///////////////////////////////////////////////////////////////////////////////
// --- Finalizar
      JU    Final_EventoRecibido_DIDO;  // Finalizar



NETWORK
TITLE = ---- Accion del Evento --> Notificacion de Cambio de Estado de Trabajo del CBOX
///////////////////////////////////////////////////////////////////////////////
///////////////////////////////////////////////////////////////////////////////
// --- Tipo CBOX
DispositivoCBOX_EventoRecibido_DIDO:NOP   0;
      L     #AtributosDeDispositivos.Numero;  // Comprobacion del numero de CCPIF
      L     100;
      /I;
      L     "CTE_OffsetCCPIF";
      -I;
      L     1;
      <>I;  // Numero de CCPIF incorrecto
      JC    Final_EventoRecibido_DIDO;

      L     #AtributosDeDispositivos.Numero;  // Calculo del numero de CBOX
      L     100;
      MOD;  // Var verlo en la DB_Dispositivos
      T     #VarTempDispositivos.Numero;

      L     #VarTempDispositivos.Numero;  // Comprobacion del numero de CBOX
      L     1;  // Es menor de 1
      <I;  // No es correcto el numero de CBOX
      JC    Final_EventoRecibido_DIDO;
      L     #VarTempDispositivos.Numero;
      L     "CTE_MaxDispositivos";  // Si es mayor que el parametro
      >I;  // No es correcto el numero de CBOX
      JC    Final_EventoRecibido_DIDO;




// ????? -------------- ?????
// ????? Por ahora nada ?????
// ????? -------------- ?????




///////////////////////////////////////////////////////////////////////////////
// --- Finalizar
      JU    Final_EventoRecibido_DIDO;



NETWORK
TITLE = ---- Accion del Evento --> Notificacion de Cambio de Estado de Trabajo de la Mesa
///////////////////////////////////////////////////////////////////////////////
///////////////////////////////////////////////////////////////////////////////
// --- Tipo Mesa
DispositivoMesa_EventoRecibido_DIDO:NOP   0;
      L     #AtributosDeDispositivos.Numero;  // Ver que mesa es
      L     "CTE_OffsetMesa";
      -I;
      T     #VarTempDispositivos.Numero;

      L     #VarTempDispositivos.Numero;  // Comprobar el numero de mesa
      L     1;  // No menor de 1
      <I;  // No es correcto
      JC    Final_EventoRecibido_DIDO;
      L     #VarTempDispositivos.Numero;
      L     "CTE_MaxMesas";  // No meyor que el parametro
      >I;  // No es correcto
      JC    Final_EventoRecibido_DIDO;




// ????? -------------- ?????
// ????? Por ahora nada ?????
// ????? -------------- ?????




///////////////////////////////////////////////////////////////////////////////
// --- Finalizar
      JU    Final_EventoRecibido_DIDO;



NETWORK
TITLE = ---- Accion del Evento --> Notificacion de Cambio de Estado de Trabajo de la Maquina
///////////////////////////////////////////////////////////////////////////////
///////////////////////////////////////////////////////////////////////////////
// --- Tipo Maquina
DispositivoMaquina_EventoRecibido_DIDO:NOP   0;
      L     #AtributosDeDispositivos.Numero;  // Ver que mesa es
      L     "CTE_OffsetMesa";
      -I;
      T     #VarTempDispositivos.Numero;

      L     #VarTempDispositivos.Numero;  // Comprobar el numero de maquina
      L     1;  // No menor de 1
      <I;  // No es correcto
      JC    Final_EventoRecibido_DIDO;
      L     #VarTempDispositivos.Numero;
      L     "CTE_MaxMesas";  // No mayor que el parametro
      >I;  // No es correcto
      JC    Final_EventoRecibido_DIDO;


///////////////////////////////////////////////////////////////////////////////
// --- Comprobar si hay Orden a la Maquina

      L     #AtributosDeDispositivos.Operacion;
      L     0;
      ==I;
      JC    Final_EstadoTrabajoDeMaquina_EventoRecibido_DIDO;

///////////////////////////////////////////////////////////////////////////////
// ---Guardar Orden para la Maquina

      L     #AtributosDeDispositivos.Operacion;  // EstadoDispo + 0 ???
      L     0;  // Orden a guardar en el DB
      +I;
      T     "DB832_Maquinas".Maquinas[#VarTempDispositivos.Numero].Operacion;


///////////////////////////////////////////////////////////////////////////////
// --- Finalizar
Final_EstadoTrabajoDeMaquina_EventoRecibido_DIDO:NOP   0;
      JU    Final_EventoRecibido_DIDO;



NETWORK
TITLE = ---- Accion del Evento --> Notificacion de Cambio de Estado de Trabajo del VTDC / ELEV
///////////////////////////////////////////////////////////////////////////////
///////////////////////////////////////////////////////////////////////////////
// --- Tipo ELEV / VTDC
Dispositivo_VTDC_ELEV_EventoRecibido_DIDO:NOP   0;
      L     #AtributosDeDispositivos.Numero;  // Ver que mesa es
      L     "CTE_OffsetMesa";
      -I;
      T     #VarTempDispositivos.Numero;

      L     #VarTempDispositivos.Numero;  // Comprobacion del numero de VTDC
      L     1;  // Es menor de 1
      <I;  // No es correcto el numero de VTDC
      JC    Final_EventoRecibido_DIDO;
      L     #VarTempDispositivos.Numero;
      L     "CTE_MaxMesas";  // Si es mayor que el parametro
      >I;  // No es correcto el numero de VTDC
      JC    Final_EventoRecibido_DIDO;


///////////////////////////////////////////////////////////////////////////////
// --- Comprobar si hay Orden a la Maquina
      L     #AtributosDeDispositivos.Operacion;
      L     0;
      ==I;
      JC    Final_EstadoTrabajoDeVTDC_EventoRecibido_DIDO;


///////////////////////////////////////////////////////////////////////////////
// ---Guardar Orden para la Maquina
      L     #AtributosDeDispositivos.Operacion;  // EstadoDispo + 0 ???
      L     0;  // Orden a guardar en el DB
      +I;
      T     "DB832_Maquinas".Maquinas[#VarTempDispositivos.Numero].VTD_ELEV.Operacion;


///////////////////////////////////////////////////////////////////////////////
// --- Operacion >>> Orden del JDT de la Posicionar el VTD
      L     #AtributosDeDispositivos.Operacion;
      L     5001;
      <>I;  // --- Hay Orden ?
      JC    Final_EstadoTrabajoDeVTDC_EventoRecibido_DIDO;


      L     #AtributosDeDispositivos.MesaHorquilla;
      T     "DB832_Maquinas".Maquinas[#VarTempDispositivos.Numero].VTD_ELEV.MesaHorquilla;
      L     #AtributosDeDispositivos.MesaCargaDesCarga;
      T     "DB832_Maquinas".Maquinas[#VarTempDispositivos.Numero].VTD_ELEV.MesaCargaDesCarga;


///////////////////////////////////////////////////////////////////////////////
// --- Finalizar
Final_EstadoTrabajoDeVTDC_EventoRecibido_DIDO:NOP   0;
      JU    Final_EventoRecibido_DIDO;



NETWORK
TITLE = ---- Final
///////////////////////////////////////////////////////////////////////////////
///////////////////////////////////////////////////////////////////////////////
///////////////////////////////////////////////////////////////////////////////
// --- Se acabo el evento
Final_EventoRecibido_DIDO:NOP   0;
      L     #P_Eventos;  // Recupero por donde voy en la lista de eventos
      LAR2;  // Regreso a buscar el siguiente evento
      JU    FinBucle_EventosRecibidos;



NETWORK
TITLE = ////////////////////////////////////////////////////////////////////////////////////////////////////////////

NETWORK
TITLE = ----

NETWORK
TITLE = Tratamiento de los EVENTOS del ROUTER
// - Inicializa variables de los atributos del Evento
// - Buscar Atributos o Final del Evento
// - Guardar datos del Evento
// 
// Mirar que atributos del Evento es ?
// - Distribuir a recoger los datos del Evento
// - Recoger el Atributo Mckey
// - Recoger el Atributo Texto a Visualizar
/////////////////////////////////////////////////////////////////////////
/////////////////////////////////////////////////////////////////////////
/////////////////////////////////////////////////////////////////////////
EventosRecibidos_Router:NOP   0;

// -- Llamar a la funcion de tratamiento de Eventos del Router
      TAR2;
      T     #P_Eventos;  // Guardo, Por donde voy en la lista de eventos

//      CALL  "FC813_EventosRec_Router"
//         NumJdT         :=#NumJDT
//         PunteroEventos :=#P_Eventos

      CALL  "FC824_Recoge_Eventos_Routing"
      ( NumJdT          := #NumJDT,
        DBEventosrouter := "ROUT_DB_Eventos_Router",
        PunteroEventos  := #P_Eventos
      );


      L     #P_Eventos;  // Recupero, Por donde voy en la lista de eventos
      LAR2;

      JU    FinBucle_EventosRecibidos;



NETWORK
TITLE = Tratamiento de los EVENTOS del QUIMAROX
// - Inicializa variables de los atributos del Evento
// - Buscar Atributos o Final del Evento
// - Guardar datos del Evento
// 
// Mirar que atributos del Evento es ?
// - Distribuir a recoger los datos del Evento
// - Recoger el Atributo Mckey
// - Recoger el Atributo Texto a Visualizar
/////////////////////////////////////////////////////////////////////////
/////////////////////////////////////////////////////////////////////////
/////////////////////////////////////////////////////////////////////////
EventosRecibidos_Quimarox:NOP   0;

// -- Llamar a la funcion de tratamiento de Eventos del Router
      TAR2;
      T     #P_Eventos;  // Guardo, Por donde voy en la lista de eventos

      CALL  "FC605_EventosRec_Quimarox"
      ( NumJdT    := #NumJDT,
        P_Eventos := #P_Eventos
      );


      L     #P_Eventos;  // Recupero, Por donde voy en la lista de eventos
      LAR2;

      JU    FinBucle_EventosRecibidos;



NETWORK
TITLE = Tratamiento de los EVENTOS del RESET de V2
// - Inicializa variables de los atributos del Evento
// - Buscar Atributos o Final del Evento
// - Guardar datos del Evento
// 
// Mirar que atributos del Evento es ?
// - Distribuir a recoger los datos del Evento
// - Recoger el Atributo Mckey
// - Recoger el Atributo Texto a Visualizar
/////////////////////////////////////////////////////////////////////////
/////////////////////////////////////////////////////////////////////////
/////////////////////////////////////////////////////////////////////////
EventosRecibidos_Reset_V2:NOP   0;

// -- Llamar a la funcion de tratamiento de Eventos del Router
      TAR2;
      T     #P_Eventos;  // Guardo, Por donde voy en la lista de eventos

      CALL  "FC814_EventosRec_Reset"
      ( NumJdT    := #NumJDT,
        P_Eventos := #P_Eventos
      );


      L     #P_Eventos;  // Recupero, Por donde voy en la lista de eventos
      LAR2;

      JU    FinBucle_EventosRecibidos;



NETWORK
TITLE = Finalizar la Funcion
// Se acabo la función
/////////////////////////////////////////////////////////////////////////
/////////////////////////////////////////////////////////////////////////
/////////////////////////////////////////////////////////////////////////
FinalizarFuncion:NOP   0;


/////////////////////////////////////////////////////////////////////////
// Limpiar el DB del UltimoRecibido del JDT01
      L     #NumJDT;
      L     1;
      <>I;
      JC    NoLimpiarDB_JDT01;

      CALL  "FC898_BorrarMensaje"
      ( DB_A_RESET := "DB807_JDT01EventosRecibidos"
      );

NoLimpiarDB_JDT01:NOP   0;

/////////////////////////////////////////////////////////////////////////
// Limpiar el DB del UltimoRecibido del JDT01
      L     #NumJDT;
      L     2;
      <>I;
      JC    NoLimpiarDB_JDT02;

      CALL  "FC898_BorrarMensaje"
      ( DB_A_RESET := "DB708_JDT02EventosRecibidos"
      );

/////////////////////////////////////////////////////////////////////////
NoLimpiarDB_JDT02:NOP   0;


/////////////////////////////////////////////////////////////////////////
NoLimpiarNada:NOP   0;


END_FUNCTION

FUNCTION "FC720_BuscarUT_EnMesa" : Void   // FC720, LAD
TITLE = "BuscarUT" - Buscar donde esta una UT determinada
{ S7_Optimized_Access := 'FALSE' }
AUTHOR : TRACKING
NAME : 20130301
VERSION : 3.0
// stored: AutoNumber false, SetENOAutomatically false
   VAR_INPUT
      Mckey : UDInt;   // Mckey de la UT
      MesaActual : UInt;   // Mesa Actual de la UT (En PLC)
   END_VAR
   VAR_OUTPUT
      NumeroUT : UInt;   // Donde esta la UT en DB_DatosUT
   END_VAR
   VAR_TEMP
      Mesa : UInt;   // Mesa
      NumUT : UInt;   // Numero UT
      ColaMckey : UInt;   // Numero de Cola de Mckey
   END_VAR
BEGIN

NETWORK
TITLE = Inicilizar
// - Iniciliza numero de DB's
// - Iniciliza variables internas
///////////////////////////////////////////////////////////////////////////////
// Inicializa las variables
      L     0;  // No existe Mckey
      T     #NumeroUT;
      T     #NumUT;

      L     #MesaActual;  // Ver que mesa es
      T     #Mesa;



NETWORK
TITLE = Bucle de la Busqueda por Mckey
// Recorre toda la cola de ordenacion de Mckey buscando la UT
// - De aqui no tiene que pasar
///////////////////////////////////////////////////////////////////////////////
///////////////////////////////////////////////////////////////////////////////
// Busqueda del Mckey en DB_OrdenadoMckey
      L     #Mckey;
      L     10000;  // 10.000 Colas de Mckey
      MOD;
      T     #ColaMckey;  // Numero de la Cola de Mckey


///////////////////////////////////////////////////////////////////////////////
      L     "DB811_ColasMckeys".Colas_Mckey[#ColaMckey].UT_PrimerMckey;
      T     #NumUT;

      L     #NumUT;
      L     0;
      ==I;
      JC    Busqueda_PorMesaActual;  // Hay UT's en la Cola de Mckey ?


///////////////////////////////////////////////////////////////////////////////
///////////////////////////////////////////////////////////////////////////////
///////////////////////////////////////////////////////////////////////////////
// Recorro las UT de la Cola de Mckey
InicoBucle_Mckey:NOP   0;
      L     "DB812_UTs_Control".UT[#NumUT].Mckey;
      L     #Mckey;  // Si es mismo MCkey
      ==D;
      JC    FinalFuncion;


///////////////////////////////////////////////////////////////////////////////
// ----- No es mismo Mckey
//       Mirar la siguiente de la Cola de Mckey
      L     "DB811_ColasMckeys".MckeyUT[#NumUT].UT_SiguienteMcKey;
      T     #NumUT;

      L     #NumUT;  // Hay mas UT's en la Cola de Mckey
      L     0;
      ==I;
      JC    Busqueda_PorMesaActual;  // No existe UT
      JU    InicoBucle_Mckey;



NETWORK
TITLE = Bucle de la Busqueda por Mesa
// Recorre toda la cola de la mesa buscando la UT
// - Si llega aqui malamente
///////////////////////////////////////////////////////////////////////////////
///////////////////////////////////////////////////////////////////////////////
///////////////////////////////////////////////////////////////////////////////
// Mirar antes de buscar si pasa Mesa
Busqueda_PorMesaActual:NOP   0;
      L     #Mesa;
      L     0;
      ==I;
      JC    Busqueda_PorListaUTs;


///////////////////////////////////////////////////////////////////////////////
///////////////////////////////////////////////////////////////////////////////
///////////////////////////////////////////////////////////////////////////////
// Empiezo a recorrer los datos de UT en la Mesa
// Miro primero si hay alguna UT en la Mesa
      L     "DB810_ColasMesas".Colas[#Mesa].UT_PrimeraMesa;
      T     #NumUT;

      L     #NumUT;
      L     0;
      ==I;
      JC    Busqueda_PorListaUTs;  // Hay UT's en la Mesa


///////////////////////////////////////////////////////////////////////////////
// Recorro las UT de las mesas
InicioBucle_MesaActual:NOP   0;
      L     "DB812_UTs_Control".UT[#NumUT].Mckey;
      L     #Mckey;  // Si es mismo MCkey
      ==D;
      JC    FinalFuncion;


///////////////////////////////////////////////////////////////////////////////
// ----- No es mismo Mckey
//       Mirar la siguinte de la Mesa
      L     "DB812_UTs_Control".UT[#NumUT].UT_SiguienteMesa;
      T     #NumUT;

      L     #NumUT;  // Hay mas UT's en la Mesa
      L     0;
      ==I;
      JC    Busqueda_PorListaUTs;  // No existe UT
      JU    InicioBucle_MesaActual;



NETWORK
TITLE = Bucle de la Busqueda por UT's directamente
// Recorre todas las UT's buscando la UT
// Si llega aqui mala cosa - muy muy malamente
///////////////////////////////////////////////////////////////////////////////
///////////////////////////////////////////////////////////////////////////////
///////////////////////////////////////////////////////////////////////////////
Busqueda_PorListaUTs:NOP   0;
      L     1;
      T     #NumUT;  // Inicializar


///////////////////////////////////////////////////////////////////////////////
// Recorro la  Lista de UTs
InicioBucle_ListaUTs:NOP   0;
      L     "DB812_UTs_Control".UT[#NumUT].Mckey;
      L     #Mckey;  // Si es mismo MCkey
      ==D;
      JC    FinalFuncion;


///////////////////////////////////////////////////////////////////////////////
// ----- No es mismo Mckey
//       Mirar la siguinte UT
      L     #NumUT;  // A la siguiente UT
      L     1;
      +I;
      T     #NumUT;

      L     #NumUT;
      L     "CTE_MaxUTs";
      >I;
      JC    FinalBucle_ListaUTs;
      JU    InicioBucle_ListaUTs;


///////////////////////////////////////////////////////////////////////////////
///////////////////////////////////////////////////////////////////////////////
///////////////////////////////////////////////////////////////////////////////
FinalBucle_ListaUTs:NOP   0;
      L     0;  // No se ha encontrado
      T     #NumUT;
      JU    FinalFuncion;



NETWORK
TITLE = Finalizar funcion
// Devuelve el Numero de UT
///////////////////////////////////////////////////////////////////////////////
///////////////////////////////////////////////////////////////////////////////
///////////////////////////////////////////////////////////////////////////////
FinalFuncion:NOP   0;
      L     #NumUT;
      T     #NumeroUT;  // Devolucion de la funcion


END_FUNCTION

FUNCTION "FC721_CrearUT_EnMesa" : Void   // FC721, LAD
TITLE = "CrearUT_EnMesa" - Crea una NUeva UT en la Mesa
{ S7_Optimized_Access := 'FALSE' }
AUTHOR : TRACKING
NAME : 20160108
VERSION : 3.2
// stored: AutoNumber false, SetENOAutomatically false
   VAR_INPUT
      McKey : UDInt;   // McKey de la UT
      MesaActual : UInt;   // Mesa Actual de la UT
   END_VAR
   VAR_OUTPUT
      NumeroUT : UInt;   // Nuemro de la UT Creada
   END_VAR
   VAR_TEMP
      Mesa : UInt;   // Mesa
      NumUT : UInt;   // Numero UT
      UTPrimera : UInt;   // UT Primera en la Mesa
      UTAnterior : UInt;   // UT Anterior en la Mesa
      UTSiguinte : UInt;   // UT Siguinte en la Mesa
      ColaMckey : UInt;   // Numnero de Cola de Ordenacion por Mckey
      TEMP_NumeroUT : UInt;
   END_VAR
BEGIN

NETWORK
TITLE = Inicilizar
// - Iniciliza numero de DB's
// - Iniciliza variables internas
////////////////////////////////////////////////////////////////////////////////
// Inicializa las variables
      L     0;  // Numero de UT Temporal
      T     #TEMP_NumeroUT;

      L     #MesaActual;  // Ver que mesa es
      T     #Mesa;



NETWORK
TITLE = Crear UT en Mesa -- Previo
////////////////////////////////////////////////////////////////////////////////
// Miro primero si hay alguna UT en la Cola de Mesa
      L     "DB810_ColasMesas".Colas[#Mesa].UT_PrimeraMesa;
      T     #UTPrimera;

      L     #UTPrimera;
      L     0;
      <>I;
      JC    HayUTs_EnColaMesa;  // Hay UT's en la Mesa
      JU    NoHayUTs_EnColaMesa;



NETWORK
TITLE = -- No Hay UT en la Cola de la Mesa
////////////////////////////////////////////////////////////////////////////////
////////////////////////////////////////////////////////////////////////////////
////////////////////////////////////////////////////////////////////////////////
// Mo hay UT's en la Cola de Mesa, Hay crear una
NoHayUTs_EnColaMesa:NOP   0;
      CALL  "FC723_InsertarUT_EnMesa"
      ( MesaActual := #MesaActual,
        NumeroUT   := #NumUT
      );

      L     0;  // NO hay Espacio para Mas UTs
      L     #NumUT;
      ==I;
      JC    Final_Funcion;


////////////////////////////////////////////////////////////////////////////////
// Ya tenemos la UT nueva, Y es la unica.
// Rellanar campos de la base de datos con lo basico
      L     #McKey;
      T     "DB812_UTs_Control".UT[#NumUT].Mckey;


      L     #MesaActual;
      L     "CTE_OffsetMesa";  // Mesa Actual Correcta
      +I;  // + Offset
      T     "DB812_UTs_Control".UT[#NumUT].MesaActual;


////////////////////////////////////////////////////////////////////////////////
// Relleno cual es la primera de la mesa
      L     #NumUT;
      T     "DB810_ColasMesas".Colas[#Mesa].UT_PrimeraMesa;

      JU    Final_EnColaMesa;



NETWORK
TITLE = -- Hay UT en la Cola de la Mesa
////////////////////////////////////////////////////////////////////////////////
////////////////////////////////////////////////////////////////////////////////
////////////////////////////////////////////////////////////////////////////////
// Hay UT's en la Cola de mesa
HayUTs_EnColaMesa:NOP   0;
      L     #UTPrimera;  // La UT Actual
      T     #NumUT;

      L     0;  // Inicio variables
      T     #UTAnterior;
      T     #UTSiguinte;


////////////////////////////////////////////////////////////////////////////////
// Empiezo a recorrer los datos de UT en la Mesa
BucleUT_EnMesa:NOP   0;

////////////////////////////////////////////////////////////////////////////////
//// CUIDADO CON ESTA CONDCION --- Se elimina
//Jose Antonio Alonso: Anulado 05/11/2015 para considerar que el MCkey 0 existe.
//porque llega el crea antes de enviar NUUT en movimientos dobles de la mesa

// "DB815_DatosUT".Datos_UTs[#NumUT].Mckey
//  L     0                           // Si es 0 es esta, la hemos creado ya
//   ==D
//   SPB MckeyCero_EnColaMesa
////////////////////////////////////////////////////////////////////////////////

      L     "DB812_UTs_Control".UT[#NumUT].UT_SiguienteMesa;
      L     0;  // Si es 0 es la ultima mesa, y hay crear una
      ==I;
      JC    FinalUT_EnColaMesa;

      L     "DB812_UTs_Control".UT[#NumUT].UT_SiguienteMesa;
      T     #NumUT;  // Mirar la siguiente de la Mesa
      JU    BucleUT_EnMesa;


////////////////////////////////////////////////////////////////////////////////
////////////////////////////////////////////////////////////////////////////////
// UT con Mckey 0, ya esta creada (NO SE UTILIZA ESTA PARTE)
MckeyCero_EnColaMesa:NOP   0;
      L     #McKey;
      T     "DB812_UTs_Control".UT[#NumUT].Mckey;

      L     #MesaActual;
      L     "CTE_OffsetMesa";  // Mesa Actual Correcta
      +I;  // + Offset
      T     "DB812_UTs_Control".UT[#NumUT].MesaActual;
      L     0;
      T     "DB812_UTs_Control".UT[#NumUT].MesaDestino;
      T     "DB812_UTs_Control".UT[#NumUT].MesaIntermedia;

      JU    Final_EnColaMesa;


////////////////////////////////////////////////////////////////////////////////
////////////////////////////////////////////////////////////////////////////////
// No hay UT con Mckey 0, hay que crear una al final de la Cola de Mesa
FinalUT_EnColaMesa:NOP   0;
      L     #NumUT;
      T     #UTAnterior;

      CALL  "FC723_InsertarUT_EnMesa"
      ( MesaActual := #MesaActual,
        NumeroUT   := #NumUT
      );

      L     0;
      L     #NumUT;
      ==I;
      JC    Final_Funcion;


////////////////////////////////////////////////////////////////////////////////
// Ya tenemos la UT nueva, Y es la unica.
// Rellanar campos de la base de datos con lo basico
      L     #UTAnterior;
      T     "DB812_UTs_Control".UT[#NumUT].UT_AnteriorMesa;

      L     #McKey;
      T     "DB812_UTs_Control".UT[#NumUT].Mckey;

      L     #MesaActual;
      L     "CTE_OffsetMesa";  // Mesa Actual Correcta
      +I;  // + Offset
      T     "DB812_UTs_Control".UT[#NumUT].MesaActual;


////////////////////////////////////////////////////////////////////////////////
// Relleno la anterior UT de la Mesa
      L     #NumUT;
      T     "DB812_UTs_Control".UT[#UTAnterior].UT_SiguienteMesa;

      JU    Final_EnColaMesa;



NETWORK
TITLE = -- Final
////////////////////////////////////////////////////////////////////////////////
////////////////////////////////////////////////////////////////////////////////
////////////////////////////////////////////////////////////////////////////////
Final_EnColaMesa:NOP   0;
      L     #NumUT;
      T     #TEMP_NumeroUT;


NETWORK
TITLE = Modificar la Ordenacion de Mckey -- Previo
////////////////////////////////////////////////////////////////////////////////
////////////////////////////////////////////////////////////////////////////////
////////////////////////////////////////////////////////////////////////////////
// Control del Mckey
      L     #McKey;  // Tiene Mckey
      L     0;
      ==D;
      JC    Final_Funcion;


////////////////////////////////////////////////////////////////////////////////
////////////////////////////////////////////////////////////////////////////////
////////////////////////////////////////////////////////////////////////////////
// Miro primero si hay alguna UT en la Cola de Mckey

      L     #McKey;
      L     10000;  // Son 10.000 las Colas de Mckey
      MOD;
      T     #ColaMckey;  // Numero de Cola de Mckey

      L     "DB811_ColasMckeys".Colas_Mckey[#ColaMckey].UT_PrimerMckey;
      T     #NumUT;

      L     #NumUT;
      L     0;
      ==I;  // No hay ninguna UT en la Cola ??????
      JC    NoHayUTs_EnColaMckey;
      JU    HayUTs_EnColaMckey;



NETWORK
TITLE = -- No Hay UT en la Cola de Ordenacion
////////////////////////////////////////////////////////////////////////////////
////////////////////////////////////////////////////////////////////////////////
////////////////////////////////////////////////////////////////////////////////
// Mo hay UT's en la Cola de Mckey
// ----- Es la primera UT de la Cola de Mckey
NoHayUTs_EnColaMckey:NOP   0;
      L     #TEMP_NumeroUT;
      T     "DB811_ColasMckeys".Colas_Mckey[#ColaMckey].UT_PrimerMckey;

      JU    Final_EnColaMcKey;



NETWORK
TITLE = -- Hay UT en la Cola de Ordenacion
////////////////////////////////////////////////////////////////////////////////
////////////////////////////////////////////////////////////////////////////////
////////////////////////////////////////////////////////////////////////////////
// Hay UT's en la Cola de Mckey
HayUTs_EnColaMckey:NOP   0;

//// CUIDADO CON ESTA CONDCION - AÑADIDO PARA INTEGRIDAD DE LA COLA DE MCKEYs
      L     #NumUT;  // Error en la Integredad de la Cola
      L     #TEMP_NumeroUT;  // Esta en la cola. IMPOSIBLE
      ==I;  // No hacer nada
      JC    Final_Funcion;


////////////////////////////////////////////////////////////////////////////////
// ---- No es la primera UT de la Cola de Mckey - Buscar cual es la ultima
BucleUT_EnColaMckey:NOP   0;
      L     #NumUT;
      T     #UTAnterior;

      L     "DB811_ColasMckeys".MckeyUT[#NumUT].UT_SiguienteMcKey;
      T     #NumUT;

      L     #NumUT;
      L     0;
      ==I;
      JC    FinalUT_EnColaMckey;  // Es la Ultima UT en la Cola ??????

//// CUIDADO CON ESTA CONDCION- AÑADIDO PARA INTEGRIDAD DE LA COLA DE MCKEYs
      L     #NumUT;  // Error en la Integredad de la Cola
      L     #TEMP_NumeroUT;  // Esta en la cola. IMPOSIBLE
      ==I;  // No hacer nada
      JC    Final_Funcion;

      JU    BucleUT_EnColaMckey;  // Continuar con la Cola de Mckey


////////////////////////////////////////////////////////////////////////////////
////////////////////////////////////////////////////////////////////////////////
////////////////////////////////////////////////////////////////////////////////
// Final de la Cola de Mckey
FinalUT_EnColaMckey:NOP   0;
      L     #TEMP_NumeroUT;  // Modificacion el la Ultima UT
      T     "DB811_ColasMckeys".MckeyUT[#UTAnterior].UT_SiguienteMcKey;

      L     #UTAnterior;  // Modificacion el la UT Creada
      T     "DB811_ColasMckeys".MckeyUT[#TEMP_NumeroUT].UT_AnteriorMckey;

      JU    Final_EnColaMcKey;



NETWORK
TITLE = --- Final
////////////////////////////////////////////////////////////////////////////////
////////////////////////////////////////////////////////////////////////////////
////////////////////////////////////////////////////////////////////////////////
// ----- No hay más final de la Ordenacion por Mckey
Final_EnColaMcKey:NOP   0;



NETWORK
TITLE = Devolucion de la Funcion
////////////////////////////////////////////////////////////////////////////////
////////////////////////////////////////////////////////////////////////////////
////////////////////////////////////////////////////////////////////////////////
Final_Funcion:NOP   0;
      L     #TEMP_NumeroUT;
      T     #NumeroUT;



END_FUNCTION

FUNCTION "FC723_InsertarUT_EnMesa" : Void   // FC723, LAD
TITLE = "InsertarUT_EnMesa" - Creacion de una UT en Mesa
{ S7_Optimized_Access := 'FALSE' }
AUTHOR : TRACKING
NAME : 20130301
VERSION : 3.0
// Mckey 0 - Y al final de la Mesa
// - Buscar una UT Libre
// - Buscar el final de la Mesa
// - Modificar datos de las UT's - Insertar
// stored: AutoNumber false, SetENOAutomatically false
   VAR_INPUT
      MesaActual : UInt;
   END_VAR
   VAR_OUTPUT
      NumeroUT : UInt;
   END_VAR
   VAR_TEMP
      NumUT : UInt;   // Numero UT
      UltimaUT : UInt;
      ValorReturn : Int;
      Cero : Byte;
   END_VAR
BEGIN

NETWORK
TITLE = Inicilizar
////////////////////////////////////////////////////////////////////////
// Inicializa las variables
      L     0;
      T     #NumeroUT;
      T     #NumUT;


///////////////////////////////////////////////////////////////////////////
///////////////////////////////////////////////////////////////////////////
///////////////////////////////////////////////////////////////////////////
/// --- Distribucion Dependiendo del Tipo de JDT (ACTUAL o VIEJO)
      SET;
      A     "Activar_JdTAntiguo";
      JC    Final_Funcion;



NETWORK
TITLE = Buscar una UT Libre
////////////////////////////////////////////////////////////////////////
////////////////////////////////////////////////////////////////////////
////////////////////////////////////////////////////////////////////////
      L     1;
      T     #NumUT;

Bucle_BuquedaUT:NOP   0;
      L     "DB812_UTs_Control".UT[#NumUT].MesaActual;
      L     0;  // Esta Vacia - 0
      ==I;
      JC    Encontrada_NuevaUT;

      L     #NumUT;  // A la siguiente UT
      L     1;
      +I;
      T     #NumUT;

      L     #NumUT;
      L     "CTE_MaxUTs";  // Si hemos llegado a la Ultima UT
      <=I;
      JC    Bucle_BuquedaUT;

      L     0;
      T     #NumUT;
      JU    Final_Funcion;



NETWORK
TITLE = UT EnContrada
////////////////////////////////////////////////////////////////////////
////////////////////////////////////////////////////////////////////////
////////////////////////////////////////////////////////////////////////
// Ya tenemos la UT nueva, Y es la unica.
// Rellanar campos de la base de datos con lo basico

Encontrada_NuevaUT:NOP   0;

////////////////////////////////////////////////////////////////////////////////
// Limpieza de la UT

      L     0;  // Valor a rellenar
      T     #Cero;

// Borrado del DB de Control de la UT
      CALL  FILL
      ( BVAL    := #Cero,
        RET_VAL := #ValorReturn,
        BLK     := "DB812_UTs_Control".UT[#NumeroUT]
      );

// Borrado del DB de la Rutas de la UT
      CALL  FILL
      ( BVAL    := #Cero,
        RET_VAL := #ValorReturn,
        BLK     := "DB813_UTs_Ruta".UT[#NumeroUT]
      );

// Borrado del DB de los Datos de la UT
      CALL  FILL
      ( BVAL    := #Cero,
        RET_VAL := #ValorReturn,
        BLK     := "DB814_UTs_Etiqueta".UT[#NumeroUT]
      );
      CALL  FILL
      ( BVAL    := #Cero,
        RET_VAL := #ValorReturn,
        BLK     := "DB815_UTs_Datos".UT[#NumeroUT]
      );
      CALL  FILL
      ( BVAL    := #Cero,
        RET_VAL := #ValorReturn,
        BLK     := "DB816_UTs_TextoPantalla".UT[#NumeroUT]
      );
      CALL  FILL
      ( BVAL    := #Cero,
        RET_VAL := #ValorReturn,
        BLK     := "DB820_UTs_DatosQUBIQA".UT[#NumeroUT]
      );
      CALL  FILL
      ( BVAL    := #Cero,
        RET_VAL := #ValorReturn,
        BLK     := "DB821_UTs_DatosIKPAL".UT[#NumeroUT]
      );


////////////////////////////////////////////////////////////////////////////////
// Relleno datos Basicos de la UT
      L     #MesaActual;  // Poner la mesa correcta
      L     "CTE_OffsetMesa";  // +Offet
      +I;
      T     "DB812_UTs_Control".UT[#NumUT].MesaActual;



NETWORK
TITLE = Colar la UT en el final de la Cola de Mesa -- Previo
////////////////////////////////////////////////////////////////////////
////////////////////////////////////////////////////////////////////////
////////////////////////////////////////////////////////////////////////
// Empiezo a recorrer los datos de UT en la Mesa
// Miro primero si hay alguna UT en la Mesa
      L     "DB810_ColasMesas".Colas[#MesaActual].UT_PrimeraMesa;
      T     #UltimaUT;

      L     #UltimaUT;
      L     0;
      <>I;  // Hay UT's en la Mesa
      JC    HayUT_EnColaMesa;
      JU    NoHayUT_EnColaMesa;



NETWORK
TITLE = No Hay UTs en la Cola de la Mesa
////////////////////////////////////////////////////////////////////////
////////////////////////////////////////////////////////////////////////
////////////////////////////////////////////////////////////////////////
// No hay ninguna, solo hay que poner cual es la primera de la mesa
NoHayUT_EnColaMesa:NOP   0;
      L     #NumUT;
      T     "DB810_ColasMesas".Colas[#MesaActual].UT_PrimeraMesa;

      JU    Final_Funcion;



NETWORK
TITLE = Hay UTs en la Cola de la Mesa
////////////////////////////////////////////////////////////////////////
////////////////////////////////////////////////////////////////////////
////////////////////////////////////////////////////////////////////////
// Si hay UT's en la mesa, hay que buscar la ultima
HayUT_EnColaMesa:NOP   0;
      L     "DB812_UTs_Control".UT[#UltimaUT].UT_SiguienteMesa;
      L     0;  // Es la Ultima
      ==I;
      JC    EncontradaUltimaUT_EnColaMesa;

      L     "DB812_UTs_Control".UT[#UltimaUT].UT_SiguienteMesa;
      T     #UltimaUT;

      JU    HayUT_EnColaMesa;


////////////////////////////////////////////////////////////////////////
// Modifico al ultima UT de la Mesa
EncontradaUltimaUT_EnColaMesa:NOP   0;
      L     #NumUT;
      T     "DB812_UTs_Control".UT[#UltimaUT].UT_SiguienteMesa;


////////////////////////////////////////////////////////////////////////
// Moodifico la nueva UT de la Mesa - Nueva Ultima

      L     #UltimaUT;
      T     "DB812_UTs_Control".UT[#NumUT].UT_AnteriorMesa;



NETWORK
TITLE = Final de la funcion
////////////////////////////////////////////////////////////////////////
////////////////////////////////////////////////////////////////////////
////////////////////////////////////////////////////////////////////////
Final_Funcion:NOP   0;

// Devolucion de la UT
      L     #NumUT;
      T     #NumeroUT;



END_FUNCTION

FUNCTION "FC898_BorrarMensaje" : Void   // FC898, LAD
{ S7_Optimized_Access := 'FALSE' }
AUTHOR : TRACKING
NAME : 20130301
VERSION : 3.0
// stored: AutoNumber false, SetENOAutomatically false
   VAR_INPUT
      DB_A_RESET : DB_ANY;
   END_VAR
   VAR_TEMP
      DESTINO : Any;
      CERO : Byte;
      BASURA : Int;
   END_VAR
BEGIN

REGION Network 1
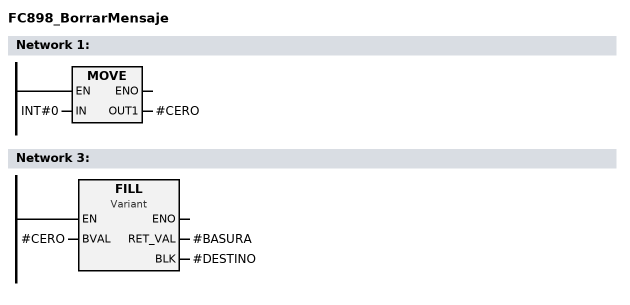
   RUNG wire#powerrail
      { S7_GenerateENO := "TRUE" } Move(in := INT#0, out1 => #CERO)
   END_RUNG
   // the same network as SCL:
   #CERO := INT#0;
END_REGION

NETWORK
TITLE = 
//ABRO EL DB PARA RESETAR Y ASI LEER SU LONGITUD
      OPN   #DB_A_RESET;
      LAR1  P##DESTINO;
// CARGAR EL ID DE SINTAXIS
      L     B#16#10;
      T     LB [AR1, P#0.0];
// CARGAR EL TIPO DE DATOS, POR DEFECTO BYTES
      L     B#16#2;
      T     LB [AR1, P#1.0];
// CARGAR LA CANTIDAD DE BYTES A COPIAR
// LEO EL TAMAÑO DEL DB A RESETAR
      L     DBLG;
      T     LW [AR1, P#2.0];
// SI ES UN DB EL ORIGEN COPIO EL NUMERO DEL DB DE DATOS
// CARGO EL NUMERO DE DB A RESETAR
      L     DBNO;
      T     LW [AR1, P#4.0];
// CARGO EL BYTE DETRABAJO
      L     0;
      SLW   3;
      T     LD [AR1, P#6.0];
// LE INDICO QUE ES UN DB
      L     B#16#84;
      T     LB [AR1, P#6.0];



REGION Network 3
   RUNG wire#powerrail
      { S7_Templates := "ptr_type := Variant" } FILL(BVAL := #CERO, RET_VAL => #BASURA, BLK => #DESTINO)
   END_RUNG
   // the same network as SCL:
   #BASURA := FILL(BVAL := #CERO, BLK => #DESTINO);
END_REGION
END_FUNCTION

FUNCTION "FC821_OrdenesDispositivos" : Void   // FC821, LAD
TITLE = "OrdenesDispositivos" - Calcular ordenes para los dispositivos
{ S7_Optimized_Access := 'FALSE' }
AUTHOR : TRACKING
NAME : 20130301
VERSION : 3.0
// - Inicializaciones
// 
// - Bucle de Dispositivos (CCPIF- CBOX)
//   - Cierre de protocolo 
//   - Busqueda de nuevo evento recibido 
//   - Tratamiento de eventos recibidos
// 
// - Bucle de Mesas (Dispositivo)
//   - Cierre de protocolo 
//   - Busqueda de nuevo evento recibido 
//   - Tratamiento de eventos recibidos
// 
// - Bucle de Maquinas (Dispositivo)
//   - Cierre de protocolo 
//   - Busqueda de nuevo evento recibido 
//   - Tratamiento de eventos recibidos
// stored: AutoNumber false, SetENOAutomatically false
   VAR_TEMP
      RecProtocoloDispositivoMesa : "UDT_ProtocoloRecDispositivo";
      P_RecProtocolo : DWord;
      P_Temporal : DWord;
      NumeroMesa : UInt;   // Numero de Mesa Actual
   END_VAR
BEGIN

NETWORK
TITLE = Inicializaciones
// Inicializacion de variables de los DB's
/////////////////////////////////////////////////////////////////////////
// --- Inicializacion de variable de los DB's



NETWORK
TITLE = Bucle de Mesas (Dipositivos)
// - Inicializacion de variables del Dispositivo (PunteroDispo y PunteroPLC)
// - Mirar si ha cerrado el protocolo
Bucle_DispositivosMesas:NOP   0;

/////////////////////////////////////////////////////////////////////////
/////////////////////////////////////////////////////////////////////////
/////////////////////////////////////////////////////////////////////////
/////////////////////////////////////////////////////////////////////////

      L     0;  // Inicializo variable, para bucle de Mesas (Dispositivos)
      T     #NumeroMesa;

/////////////////////////////////////////////////////////////////////////
// --- Empieza el recorrido por todos los dispositivos
InicioBucle_DispositivosMesa:NOP   0;
      L     #NumeroMesa;  // Incremento en uno el numero de Mesa
      L     1;
      +I;
      T     #NumeroMesa;

/////////////////////////////////////////////////////////////////////////
// Ya he recorrido todos las Mesas (Dispositivos) ?
      L     #NumeroMesa;  // Ya estan todas las Mesas (Dispositivos)
      L     "CTE_MaxMesas";
      >I;  // Ir a Maquinas (Dispositivos)
      JC    FinalFuncion;


/////////////////////////////////////////////////////////////////////////
/// Mirar Si hay Mesa Configurada (2019 / 01 /18)
      SET;

      AN    "DB850_DefinicionMesas".Mesa[#NumeroMesa].ConfigMesa.MesaPaso;
      AN    "DB850_DefinicionMesas".Mesa[#NumeroMesa].ConfigMesa.MesaCruce;
      AN    "DB850_DefinicionMesas".Mesa[#NumeroMesa].ConfigMesa.MesaMultiplesDestinos;
      AN    "DB850_DefinicionMesas".Mesa[#NumeroMesa].ConfigMesa.MesaTL;
      JC    InicioBucle_DispositivosMesa;


/////////////////////////////////////////////////////////////////////////
// --- Recoger Datos del Dispositivo (Protocolo)
      CALL  MOVE
      ( IN  := "DB841_Recepcion".DispoMesa[#NumeroMesa].Protocolo,
        OUT := #RecProtocoloDispositivoMesa
      );

      L     P##RecProtocoloDispositivoMesa;
      T     #P_RecProtocolo;



/////////////////////////////////////////////////////////////////////////
// --- Mirar si esta cerrado el protocolo
      L     "DB831_Mesas".Mesas[#NumeroMesa].EstadoOrdenDispo;
      L     0;  // Mirar si no esta Cerrado el Protocolo ?
      <>I;  // Ir a Cerrar Protocolo de la Mesa (Dispositivo)
      JC    CerrarProtocolo_DispositivosMesa;


/////////////////////////////////////////////////////////////////////////
// Ir a Buscar Evento Nuevo para la Mesa (Dispositivo)
      JU    TratarEventosRecibidos_DispositivosMesa;



NETWORK
TITLE = Cierre del Protocolo de Mesas (Dispositivos)
// - Recoger como esta el RecepOK
// - Distribuir dependiendo del Status del Protocolo
//   - Esta en Fase 1 - Esperando que se desactive RecepOK 
//   - Esta en Fase 2 - Esperando que se active RecepOK
CerrarProtocolo_DispositivosMesa:NOP   0;

/////////////////////////////////////////////////////////////////////////
/////////////////////////////////////////////////////////////////////////
/////////////////////////////////////////////////////////////////////////
/////////////////////////////////////////////////////////////////////////
// --- Distribuir dependiendo el Status del Protocolo

      L     "DB831_Mesas".Mesas[#NumeroMesa].EstadoOrdenDispo;
      L     1;  // Mirar en que Fase esta el Protocolo?
      ==I;  // Protocolo - Esta en Fase 1
      JC    ProtocoloEnFase_01_DispositivoMesa;

// Protocolo - Esta en Fase 2
      JU    ProtocoloEnFase_02_DispositivoMesa;


/////////////////////////////////////////////////////////////////////////
/////////////////////////////////////////////////////////////////////////
// --- Fase 1 - Esperando que se Desactive RecepOK del Dispositivo
ProtocoloEnFase_01_DispositivoMesa:NOP   0;
      SET;  // DesActivado la RecepOK ?
      A     "DB840_Emision".DispoMesa[#NumeroMesa].Protocolo.RecepOK;
      JC    FinCerrarProtocolo_DispositivosMesa;


// Fase 0 - Acabado el Protocolo
      L     0;
      T     "DB831_Mesas".Mesas[#NumeroMesa].EstadoOrdenDispo;

      JU    FinCerrarProtocolo_DispositivosMesa;


/////////////////////////////////////////////////////////////////////////
/////////////////////////////////////////////////////////////////////////
// --- Fase 2 - Esperando que se active RecepOK del Dispositivo
ProtocoloEnFase_02_DispositivoMesa:NOP   0;
      SET;  // Activado la RecepOK ?
      AN    "DB840_Emision".DispoMesa[#NumeroMesa].Protocolo.RecepOK;
      JC    FinCerrarProtocolo_DispositivosMesa;


// Fase 1 - Espnierando que desactive el RecpOK
      L     1;
      T     "DB831_Mesas".Mesas[#NumeroMesa].EstadoOrdenDispo;

      L     LW [#P_RecProtocolo];
      L     W#16#80;
      AW;  // Desactivo la Orden enviada
      T     LW [#P_RecProtocolo];

      CALL  MOVE
      ( IN  := #RecProtocoloDispositivoMesa,
        OUT := "DB841_Recepcion".DispoMesa[#NumeroMesa].Protocolo
      );

      L     0;  // Borrar Words Auxiliares
      T     "DB841_Recepcion".DispoMesa[#NumeroMesa].Auxiliar_01;
      T     "DB841_Recepcion".DispoMesa[#NumeroMesa].Auxiliar_02;
      T     "DB841_Recepcion".DispoMesa[#NumeroMesa].Auxiliar_03;
      T     "DB841_Recepcion".DispoMesa[#NumeroMesa].ORDE;

      JU    FinCerrarProtocolo_DispositivosMesa;


/////////////////////////////////////////////////////////////////////////
/////////////////////////////////////////////////////////////////////////
// --- Final del Segmento del Cierre de Protocolo
FinCerrarProtocolo_DispositivosMesa:NOP   0;
// Finalizar, ir al Siguiente Dispositivo
      JU    InicioBucle_DispositivosMesa;



NETWORK
TITLE = Busqueda de nuevo evento para las Mesas (Dispositivo)
// - Pasos a seguir:
//   - Mirar si se puede tratar el evento recibido
//   - Mirar si hay algun evento recibido
//   - Distribucion de los eventos recibidos
TratarEventosRecibidos_DispositivosMesa:NOP   0;

/////////////////////////////////////////////////////////////////////////
/////////////////////////////////////////////////////////////////////////
/////////////////////////////////////////////////////////////////////////
/////////////////////////////////////////////////////////////////////////
// -- Condiciones para enviar alguna orden:
//    - StatusEmisino = 0
//    - StatusRecepcion <> 0
//

/////////////////////////////////////////////////////////////////////////
// --- Mirar si se puede Enviar orden (StatusEmision = 0)
      L     "DB831_Mesas".Mesas[#NumeroMesa].EstadoEmisionEvento;
      L     0;  // Esta emitido todo (Eventos)
      <>I;  // No se puede enviar orden
      JC    FinEventosRecibidos_DispositivosMesa;

/////////////////////////////////////////////////////////////////////////
// --- Mirar si hay algo que Enviar (StatusRecepcion <> 0)
      L     "DB831_Mesas".Mesas[#NumeroMesa].EstadoRecepcionEvento;
      L     0;  // Ha recibido algun Evento ?
      ==I;  // No Ha recibido Ninguno
      JC    FinEventosRecibidos_DispositivosMesa;


/////////////////////////////////////////////////////////////////////////
/////////////////////////////////////////////////////////////////////////
/////////////////////////////////////////////////////////////////////////
// --- Distribucion para el Tratamiento del Evento Recibido

/////////////////////////////////////////////////////////////////////////
// --- Peticion de Refresco de Datos del Dispositivo
      L     "DB831_Mesas".Mesas[#NumeroMesa].EstadoRecepcionEvento;
      L     250;
      ==I;
      JC    RefrescoDatosEventosRecibidos_DispositivosMesa;


/////////////////////////////////////////////////////////////////////////
// --- Nuevo Estado del Dispositivo >>> Sin Orden
      L     "DB831_Mesas".Mesas[#NumeroMesa].EstadoRecepcionEvento;
      L     260;
      ==I;
      JC    RefrescoDatosEventosRecibidos_DispositivosMesa;


/////////////////////////////////////////////////////////////////////////
// --- Solo queda este tipo de evento: 260...274  (Nuevo Estado del Dispositivo)
      L     "DB831_Mesas".Mesas[#NumeroMesa].EstadoRecepcionEvento;
      L     261;
      <I;  // < 260 ? - No es Nuevo Estado
      JC    DefectoEventosRecibidos_DispositivosMesa;
      L     "DB831_Mesas".Mesas[#NumeroMesa].EstadoRecepcionEvento;
      L     274;
      >I;  // > 274 ? - No es Nuevo Estado
      JC    DefectoEventosRecibidos_DispositivosMesa;

/////////////////////////////////////////////////////////////////////////
// Si es Nuevo Estado
      JU    NuevoEstadoEventosRecibidos_DispositivosMesa;


/////////////////////////////////////////////////////////////////////////
/////////////////////////////////////////////////////////////////////////
/////////////////////////////////////////////////////////////////////////
// --- Dar por tratada, no esta programado este Evento recibido
DefectoEventosRecibidos_DispositivosMesa:NOP   0;
      L     0;  // Darlo por tratado
      T     "DB831_Mesas".Mesas[#NumeroMesa].EstadoRecepcionEvento;

      JU    FinEventosRecibidos_DispositivosMesa;


/////////////////////////////////////////////////////////////////////////
/////////////////////////////////////////////////////////////////////////
/////////////////////////////////////////////////////////////////////////
// --- Final del Segmento de Buscar Nuevo Evento
FinEventosRecibidos_DispositivosMesa:NOP   0;
// Finalizar, ir al Siguiente Dispositivo
      JU    InicioBucle_DispositivosMesa;



NETWORK
TITLE = Tratamiento de los eventos para las Mesas (Dispositivos)
// - Lista de Eventos Recibidos
//   - Evento de Peticion de Refresco de datos
//   - Evento de Nuevo Estado
/////////////////////////////////////////////////////////////////////////
/////////////////////////////////////////////////////////////////////////
/////////////////////////////////////////////////////////////////////////
// --- Evento de Peticion de Refresco de Datos del Dispositivo
//     * Mirar si EstadoGeneral esta libre
//     * Darlo por tratado
//       Activacion de Generacion del Evento de Peticion de Refresco
RefrescoDatosEventosRecibidos_DispositivosMesa:NOP   0;
      L     "DB831_Mesas".Mesas[#NumeroMesa].EstadoGeneralEvento;
      L     0;  // EstadoGeneral - Libre
      <>I;
      JC    FinEventosRecibidos_DispositivosMesa;

/////////////////////////////////////////////////////////////////////////
// --- Darlo por tratado y Activacion de Generacion de Evento
      L     25;  // 25 - Refresco de Datos del dispositivo
      T     "DB831_Mesas".Mesas[#NumeroMesa].EstadoGeneralEvento;
      L     0;  // Darlo por tratado
      T     "DB831_Mesas".Mesas[#NumeroMesa].EstadoRecepcionEvento;

/////////////////////////////////////////////////////////////////////////
// --- Fin Evento de Peticion de Refresco de Datos del Dispositivo
      JU    FinEventosRecibidos_DispositivosMesa;


/////////////////////////////////////////////////////////////////////////
/////////////////////////////////////////////////////////////////////////
/////////////////////////////////////////////////////////////////////////
// --- Evento de Nuevo Estado del Dispositivo
//     * Calculo del Nuevo Estado Recibido
//     * Activar Nuevo Estado
//     * Darlo por tratado este Evento
//       Activar Protocolo del Dispositivo

/////////////////////////////////////////////////////////////////////////
// --- Calcula del Nuevo Estado Recibido
NuevoEstadoEventosRecibidos_DispositivosMesa:NOP   0;
      L     "DB831_Mesas".Mesas[#NumeroMesa].EstadoRecepcionEvento;
      L     260;
      -I;  // Numero de Bit a Activar
      L     #P_RecProtocolo;
      +D;  // Direccion del Bit a Activar
      T     #P_Temporal;

/////////////////////////////////////////////////////////////////////////
// --- Activar Orden Recibida (Nuevo Estado)

      SET;  // Poner a '1' el bit de la orden
      S     L [#P_Temporal];  // Orden del PLC calculada

      CALL  MOVE
      ( IN  := #RecProtocoloDispositivoMesa,
        OUT := "DB841_Recepcion".DispoMesa[#NumeroMesa].Protocolo
      );

/////////////////////////////////////////////////////////////////////////
// --- Darlo por tratado y Activar Protocolo
      L     2;  // Fase 2 - Esperando que active el RecepOK
      T     "DB831_Mesas".Mesas[#NumeroMesa].EstadoOrdenDispo;
      L     0;  // Darlo por tratado
      T     "DB831_Mesas".Mesas[#NumeroMesa].EstadoRecepcionEvento;


/////////////////////////////////////////////////////////////////////////
// --- Fin Evento de Nuevo Estado del Dispositivo
      JU    FinEventosRecibidos_DispositivosMesa;



NETWORK
TITLE = Final de la funcion
// Se acabo
FinalFuncion:NOP   0;

END_FUNCTION

FUNCTION "FC811_EventosGenerados" : Void   // FC811, LAD
TITLE = "EventosGenerados" - Se generar la lista de Eventos a Emitir
{ S7_Optimized_Access := 'FALSE' }
AUTHOR : TRACKING
NAME : 20160407
VERSION : 4.2
// - Inicializaciones
// - Mirar si se pueden generar eventos
// - Generar eventos de las UT's
// - Generar eventos de los dispositivos
// - Generar eventos de las Mesas
// stored: AutoNumber false, SetENOAutomatically false
   VAR_INPUT
      NumJdT : UInt;
   END_VAR
   VAR_TEMP
      DBEventos : Word;   // Num. DB de eventos generados
      NumDBEventos : UInt;
      P_Eventos : DWord;   // Puntero al DB de Eventos Generados
      MaxBytes : UInt;
      InicioBucleMesas : UInt;
      FinalBucleMesas : UInt;
      NumBytes : UInt;   // Numero de Bytes a Emitir
      P_Temporal : DWord;
      NumMesa : UInt;   // Numero de Mesa a mirar
      IndiceEtiqueta : UInt;
      NumeroUT : UInt;   // Numero de UT a mirar
      EventoUT : UInt;   // Numero de Evento Generado en la UT
      EventoDispositivo : UInt;   // Numero de Evento Genarado en el Dispositivo
      NivelPantalla : UInt;   // Numero de nivel de pantalla
      Convertir : UInt;
      Conversion : DWord;
      Valor : UDInt;
      Offset : UInt;
      Proceso : UInt;
      ResultadoProceso : UInt;
      ValorReturn : Int;
      MesaDeJDT02 : Bool;
      JDT02_Activo : Bool;
      DispoDeJDT02 : Bool;
   END_VAR
BEGIN

NETWORK
TITLE = Inicializaciones
// - Inicializar las variables de los DB's
////////////////////////////////////////////////////////////////////////////////
////////////////////////////////////////////////////////////////////////////////
/// Inicio Que conexion es de JDT

      SET;
      R     #JDT02_Activo;
      L     "JDT1_NDB_EventosEmi";
      T     #DBEventos;
      T     #NumDBEventos;
      L     "JDT2_MaxBytes";
      T     #MaxBytes;

      L     "JDT1_InicioBucleMesas";  // Tamaño Bucles
      T     #InicioBucleMesas;
      L     "JDT1_FinalBucleMesas";
      T     #FinalBucleMesas;

      L     #NumJdT;
      L     2;
      <>I;
      JC    NoJDT02;

      SET;
      S     #JDT02_Activo;
      L     "JDT2_NDB_EventosEmi";
      T     #DBEventos;
      T     #NumDBEventos;
      L     "JDT2_MaxBytes";
      T     #MaxBytes;

      L     "JDT2_InicioBucleMesas";  // Tamaño Bucles
      T     #InicioBucleMesas;
      L     "JDT2_FinalBucleMesas";
      T     #FinalBucleMesas;

NoJDT02:NOP   0;

/// FIn Que conexion es de JDT
////////////////////////////////////////////////////////////////////////////////
////////////////////////////////////////////////////////////////////////////////



NETWORK
TITLE = Mirar si se pueden generar eventos
// - Inicializo el Numero de Bytes y el puntero del DB de Eventos Generados
// - Calcula el Tamaño de bytes que hay en el DB de Eventos Genardos
// - Comprobamos si hay sitio para Eventos
////////////////////////////////////////////////////////////////////////////////
// Inicializo el Numero de Bytes y el puntero del DB Eventos Generados

      L     0;
      T     #NumBytes;  // Inicializo el numero de Bytes
      LAR2;  // Inicializo el puntero de Eventos Generados

////////////////////////////////////////////////////////////////////////////////
// Calcula el tamaño de bytes que hay en el DB Eventos Generados

      OPN   DB [#DBEventos];

InicioBucleBusquedaFin_BufferEventos:NOP   0;
      L     DBB [AR2, P#0.0];
      L     0;
      ==I;
      JC    FinBucleBusquedaFin_BufferEventos;  // Buscamos el final del DB = 0

      +AR2  P#1.0;
      JU    InicioBucleBusquedaFin_BufferEventos;

FinBucleBusquedaFin_BufferEventos:NOP   0;
      TAR2;  // Guardo el puntero
      T     #P_Eventos;  // Sacamos el NumBytes Escritos
      SRD   3;
      T     #NumBytes;

////////////////////////////////////////////////////////////////////////////////
// Comprobamos si hay sitio para mas Eventos

      L     #NumBytes;  // Miramos si hay sitio
      L     #MaxBytes;  // Max. que se pueden emitir, parametro
      >I;
      JC    FinalFuncion;  // No se pueden generar más eventos



NETWORK
TITLE = Generar Eventos de las UT's
// - Recorrer todas las Mesas Buscando UT'que necesiten generar Eventos
//   Dos bucles anidados Mesas y UT's dentro de las Mesas ( No se hace)
// - Recorrer todas las UT's (Se hace
////////////////////////////////////////////////////////////////////////////////
////////////////////////////////////////////////////////////////////////////////
////////////////////////////////////////////////////////////////////////////////
// Recorrer todas las Mesas

      L     #InicioBucleMesas;
      T     #NumMesa;

InicioBucleMesa_EventosUT:NOP   0;
////////////////////////////////////////////////////////////////////////////////
/// Mirar Si pertenece al JDT

      SET;
      X     "DB850_DefinicionMesas".Mesa[#NumMesa].ConfigMesa.MesaDeJDT02;
      XN    #JDT02_Activo;  // JDT01 o JDT02 ?
      =     #MesaDeJDT02;

      SET;
      AN    #MesaDeJDT02;
      JC    ContinuarBucleMesa_EventosUT;

////////////////////////////////////////////////////////////////////////////////
// Mirar si esta definido como mesa de tracking

      SET;
      AN    "DB850_DefinicionMesas".Mesa[#NumMesa].ConfigMesa.MesaPaso;
      AN    "DB850_DefinicionMesas".Mesa[#NumMesa].ConfigMesa.MesaCruce;
      AN    "DB850_DefinicionMesas".Mesa[#NumMesa].ConfigMesa.MesaMultiplesDestinos;
      JC    ContinuarBucleMesa_EventosUT;


////////////////////////////////////////////////////////////////////////////////

      L     "DB810_ColasMesas".Colas[#NumMesa].UT_PrimeraMesa;
      T     #NumeroUT;

      L     #NumeroUT;
      L     0;
      ==I;
      JC    ContinuarBucleMesa_EventosUT;  // No hay UT's en la Mesa


////////////////////////////////////////////////////////////////////////////////
// --- Recorrer todas las UT's de la Mesa
InicioBucleUT_EventosUT:NOP   0;

      L     "DB812_UTs_Control".UT[#NumeroUT].EstadoEventoAGenerar;
      T     #EventoUT;  // Para ver si hay Evento de UT

      L     #EventoUT;  // Mirar si hay evento a generar
      L     100;
      >=I;
      JC    Generar_EventosUT;  // Si es >= 100 Hay evento a generar


////////////////////////////////////////////////////////////////////////////////
ContinuarBucleUT_EventosUT:NOP   0;
      L     "DB812_UTs_Control".UT[#NumeroUT].UT_SiguienteMesa;
      T     #NumeroUT;

      L     #NumeroUT;
      L     0;
      ==I;
      JC    ContinuarBucleMesa_EventosUT;  // No hay mas UT's en la Mesa

      JU    InicioBucleUT_EventosUT;  // Seguir recorriendo la Mesa


////////////////////////////////////////////////////////////////////////////////
// --- Continuar recorriendo el resto de Mesas
ContinuarBucleMesa_EventosUT:NOP   0;
      L     #NumMesa;
      L     #FinalBucleMesas;
      >=I;
      JC    EventosMesa;  // Ya no hay más UT's, recorrer dispositivos

      L     #NumMesa;  // +1, Para la Siguiente UT
      L     1;
      +I;
      T     #NumMesa;

      JU    InicioBucleMesa_EventosUT;  // Ir a mirar la siguiente UT


////////////////////////////////////////////////////////////////////////////////
// Comprobacion del tamaño del DB de Eventos Generados
FinBucles_EventosUT:NOP   0;
      TAR2;
      T     #P_Eventos;
      SRD   3;
      T     #NumBytes;

      L     #NumBytes;  // Miramos si hay sitio
      L     #MaxBytes;
      >I;
      JC    FinalFuncion;  // No se pueden generar más eventos
      JU    ContinuarBucleUT_EventosUT;  // Seguir con las UT's



NETWORK
TITLE = Formatear Eventos de las UTs - Distribucion
Generar_EventosUT:NOP   0;

////////////////////////////////////////////////////////////////////////////////
////////////////////////////////////////////////////////////////////////////////
// -- Formateo del Evento LOCA - Diferentes Motivos (Normal, Reset, Galibo ...)
// -- Formateo del Evento RUT? - Diferentes (Reset, PLC, ...)
// -- Formateo del Evento RET! - Ausencia de la Mesa
// -- Formateo del Evento BOR! - Borrada UT del Sistema
// -- Formateo del Evento DATO - Refresco de Datos de la UT
// -- Formateo del Evento NUUT - Nueva UT en la Mesa
// -- Formateo del Evento DAT? - Peticion de Datos para la UT
// -- Formateo del Evento PEMB (Peticion de Datos de Embandejado de la UT)
////////////////////////////////////////////////////////////////////////////////
////////////////////////////////////////////////////////////////////////////////
// Distribucion para Eventos de las UT's

      L     #EventoUT;  // Formateo del evento
      L     100;  // Presencia Normal
      ==I;
      JC    GenerarEvento_LOCA_EventosUT;

      L     #EventoUT;  // Formateo del evento
      L     101;  // Presencia de Reset
      ==I;
      JC    GenerarEvento_LOCA_EventosUT;

      L     #EventoUT;  // Formateo del evento
      L     102;  // Presencia de Galibo
      ==I;
      JC    GenerarEvento_LOCA_EventosUT;

      L     #EventoUT;  // Formateo del evento
      L     103;  // Ausencia
      ==I;
      JC    GenerarEvento_RET_EventosUT;

      L     #EventoUT;  // Formateo del evento
      L     110;  // Refresco de datos de la UT
      ==I;
      JC    GenerarEvento_DATO_EventoUT;

      L     #EventoUT;  // Formateo del evento
      L     121;  // Peticion de Ruta por MOTIVO --> Reset
      ==I;
      JC    GenerarEvento_RUT_EventoUT;

      L     #EventoUT;  // Formateo del evento
      L     122;  // Peticion de Ruta por MOTIVO --> Bloqueo
      ==I;
      JC    GenerarEvento_RUT_EventoUT;

      L     #EventoUT;  // Formateo del evento
      L     123;  // Peticion de Ruta por MOTIVO --> Llegada a su Destino
      ==I;
      JC    GenerarEvento_RUT_EventoUT;

      L     #EventoUT;  // Formateo del evento
      L     124;  // Peticion de Ruta por MOTIVO --> No tiene Destino
      ==I;
      JC    GenerarEvento_RUT_EventoUT;

      L     #EventoUT;  // Formateo del evento
      L     125;  // Peticion de Ruta por MOTIVO --> Fuera de Ruta
      ==I;
      JC    GenerarEvento_RUT_EventoUT;

      L     #EventoUT;  // Formateo del evento
      L     126;  // Peticion de Ruta por MOTIVO --> Robo de Garra a Elevador
      ==I;
      JC    GenerarEvento_RUT_EventoUT;

      L     #EventoUT;  // Formateo del evento
      L     131;  // Borrar la UT de la Base de datos
      ==I;
      JC    GenerarEvento_BOR_EventosUT;

      L     #EventoUT;  // Formateo del evento
      L     132;  // Nueva UT en la BD
      ==I;
      JC    GenerarEvento_NUUT_EventosUT;

      L     #EventoUT;  // Formateo del evento
      L     141;  // Peticion de datos para la UT
      ==I;
      JC    GenerarEvento_DAT_EventosUT;

      L     #EventoUT;  // Formateo del evento
      L     145;  // Chequeo de la UT >>> Por Reset
      ==I;
      JC    GenerarEvento_CHE_EventosUT;

      L     #EventoUT;  // Formateo del evento     // Fecha 2019 01 18
      L     161;  // Peticion de datos de Embandejado para la UT
      ==I;
      JC    GenerarEvento_PEMB_EventosUT;


////////////////////////////////////////////////////////////////////////////////
////////////////////////////////////////////////////////////////////////////////
////////////////////////////////////////////////////////////////////////////////
// --- Dar por formateado el Evento

      L     0;  // 0 - Dar por Tratado
      T     "DB812_UTs_Control".UT[#NumeroUT].EstadoEventoAGenerar;

      JU    FinBucles_EventosUT;

// Fin de la distribucion para generar los eventos
////////////////////////////////////////////////////////////////////////////////
////////////////////////////////////////////////////////////////////////////////
////////////////////////////////////////////////////////////////////////////////



NETWORK
TITLE = ---- Eventos de UT - Esta en Mesa - LOCA
// - Distribucion para Eventos de las UT's
// - Formateo de Eventos
//   - Evento LOCA (Cambio de Mesa de la UT
//   - Evento RUT? (Petición de Ruta para la UT)
//   - Evento NUUT (Nueva UT en la instalacion)
//   - Evento DATO (Cambio de de datos de la UT)
//   - Evento BOR! (UT Borrada de la Base de datos)
//   - Evento DAT? (Peticion de datos de la UT)
//   - Evento RET! (Retirada de la UT)
GenerarEvento_LOCA_EventosUT:NOP   0;

////////////////////////////////////////////////////////////////////////////////
////////////////////////////////////////////////////////////////////////////////
////////////////////////////////////////////////////////////////////////////////
// -- Formateo del Evento LOCA - Diferentes Motivos (Normal, Reset, Galibo ...)

      L     #P_Eventos;
      LAR2;  // Puntero al DB de Eventos Generados

      TAR2;  // Mirar si es el primer evento de la lista
      L     0;
      ==I;
      JC    InicioBuffer_LOCA_EventosUT;  // Es el primero

      OPN   DB [#DBEventos];  // Hay que añadir si no es el primer evento
      L     ',';  // Separador entre eventos ','
      T     DBB [AR2, P#0.0];
      +AR2  P#1.0;

InicioBuffer_LOCA_EventosUT:NOP   0;
      OPN   DB [#DBEventos];  // DB de Eventos Generados (A Emitir)
      L     '{';  // Inicio de Evento '{'
      T     DBB [AR2, P#0.0];
      +AR2  P#1.0;


////////////////////////////////////////////////////////////////////////////////
      L     'LOCA';  // Evento 'LOCA'
      T     DBD [AR2, P#0.0];
      +AR2  P#4.0;

      L     '[';  // Evento - Atributo Mckey '[MCKY]'
      T     DBB [AR2, P#0.0];
      L     'MCKY';
      T     DBD [AR2, P#1.0];
      L     ']';  // Evento - Atributo Mckey '[MCKY]'
      T     DBB [AR2, P#5.0];
      +AR2  P#6.0;

      L     "DB812_UTs_Control".UT[#NumeroUT].Mckey;
      T     #Valor;

// --- Convertir Valor a ASCII - Mckey
      TAR2;
      SRD   3;
      T     #NumBytes;  // Miro que offset tiene la String

      CALL  "FC893_Obtener_StringDelAtributo"
      ( DB_String := #NumDBEventos,
        OffsetIni := #NumBytes,
        Valor     := #Valor,
        OffsetFin := #Offset
      );  // Llamo a ObtenerStrinAtributo

      L     #Offset;
      SLD   3;
      LAR2;  // Recupero que offset tiene la String

// --- Ya esta convertido el Valor a ASCI - Fin Mckey


////////////////////////////////////////////////////////////////////////////////
      OPN   DB [#DBEventos];
      L     '[';  // Evento - Atributo Mesa Actual '[MESA]'
      T     DBB [AR2, P#0.0];
      L     'MESA';
      T     DBD [AR2, P#1.0];
      L     ']';
      T     DBB [AR2, P#5.0];
      +AR2  P#6.0;

      L     "DB812_UTs_Control".UT[#NumeroUT].MesaActual;
      T     #Valor;

// --- Convertir Valor a ASCII -  Mesa Actual
      TAR2;
      SRD   3;
      T     #NumBytes;  // Miro que offset tiene la String

      CALL  "FC893_Obtener_StringDelAtributo"
      ( DB_String := #NumDBEventos,
        OffsetIni := #NumBytes,
        Valor     := #Valor,
        OffsetFin := #Offset
      );  // Llamo a ObtenerStrinAtributo

      L     #Offset;
      SLD   3;
      LAR2;  // Recupero que offset tiene la String

// --- Ya esta convertido el Valor a ASCI - Fin Mesa Actual


////////////////////////////////////////////////////////////////////////////////
// --- Final del Formateo del Evento ---

      OPN   DB [#DBEventos];  // DB de Eventos Generados (A Emitir)
      L     '}';  // Fin de Evento '}'
      T     DBB [AR2, P#0.0];
      +AR2  P#1.0;



////////////////////////////////////////////////////////////////////////////////
////////////////////////////////////////////////////////////////////////////////
////////////////////////////////////////////////////////////////////////////////
// --- Dar por formateado el Evento

      L     0;  // 0 - Dar por Tratado
      T     "DB812_UTs_Control".UT[#NumeroUT].EstadoEventoAGenerar;

////////////////////////////////////////////////////////////////////////////////
/// Hay que Pedir Datos
      SET;
      AN    "DB812_UTs_Control".UT[#NumeroUT].AtributosDeLaUT.PeticionDeDatos;
      JC    NoPedirDatos_LOCA_EventosUT;

      L     141;
      T     "DB812_UTs_Control".UT[#NumeroUT].EstadoEventoAGenerar;

NoPedirDatos_LOCA_EventosUT:NOP   0;

////////////////////////////////////////////////////////////////////////////////
/// Hay que Generar mas Eventos
      L     #EventoUT;  // Formateo del evento
      L     100;  // Presencia Normal
      ==I;
      JC    FinBucles_EventosUT;

////////////////////////////////////////////////////////////////////////////////
/// Es de Reset de Pantalla, Auto Generar Nuevo Evento
      L     121;  // 121 - Generar evento de Pedir Ruta (Por Reset)
      T     "DB812_UTs_Control".UT[#NumeroUT].EstadoEventoAGenerar;

      L     #EventoUT;  // Formateo del evento
      L     101;  // Presencia de Reset
      ==I;
      JC    FinBucles_EventosUT;


////////////////////////////////////////////////////////////////////////////////
/// Es de Galibo, Auto Generar Nuevo Evento
      L     110;  // Enviar datos de UT
      T     "DB812_UTs_Control".UT[#NumeroUT].EstadoEventoAGenerar;

      JU    FinBucles_EventosUT;

// Fin del Evento LOCA
////////////////////////////////////////////////////////////////////////////////
////////////////////////////////////////////////////////////////////////////////
////////////////////////////////////////////////////////////////////////////////



NETWORK
TITLE = ---- Evento de UT - Peticion de Ruta - RUT?
GenerarEvento_RUT_EventoUT:NOP   0;

////////////////////////////////////////////////////////////////////////////////
////////////////////////////////////////////////////////////////////////////////
////////////////////////////////////////////////////////////////////////////////
////////////////////////////////////////////////////////////////////////////////
// -- Formateo del Evento RUT? - Diferentes (Reset, PLC, ...)

      L     #P_Eventos;
      LAR2;  // Puntero al DB de Eventos Generados

      TAR2;  // Mirar si es el primer evento de la lista
      L     0;
      ==I;
      JC    InicioBuffer_RUT_EventosUT;  // Es el primero

      OPN   DB [#DBEventos];  // Hay que añadir si no es el primer evento
      L     ',';  // Separador entre eventos ','
      T     DBB [AR2, P#0.0];
      +AR2  P#1.0;

InicioBuffer_RUT_EventosUT:NOP   0;
      OPN   DB [#DBEventos];  // DB de Eventos Generados (A Emitir)
      L     '{';  // Inicio de Evento '{'
      T     DBB [AR2, P#0.0];
      +AR2  P#1.0;

      L     'RUT?';  // Evento 'RUT?'
      T     DBD [AR2, P#0.0];
      +AR2  P#4.0;


////////////////////////////////////////////////////////////////////////////////
      L     '[';  // Evento - Atributo Mckey '[MCKEY]'
      T     DBB [AR2, P#0.0];
      L     'MCKY';
      T     DBD [AR2, P#1.0];
      L     ']';
      T     DBB [AR2, P#5.0];
      +AR2  P#6.0;

      L     "DB812_UTs_Control".UT[#NumeroUT].Mckey;
      T     #Valor;

// --- Convertir Valor a ASCII - Mckey
      TAR2;
      SRD   3;
      T     #NumBytes;  // Miro que offset tiene la String

      CALL  "FC893_Obtener_StringDelAtributo"
      ( DB_String := #NumDBEventos,
        OffsetIni := #NumBytes,
        Valor     := #Valor,
        OffsetFin := #Offset
      );  // Llamo a ObtenerStrinAtributo

      L     #Offset;
      SLD   3;
      LAR2;  // Recupero que offset tiene la String

// --- Ya esta convertido el Valor a ASCI - Fin Mckey


////////////////////////////////////////////////////////////////////////////////
      OPN   DB [#DBEventos];
      L     '[';  // Evento - Atributo Mesa Actual '[MESA]'
      T     DBB [AR2, P#0.0];
      L     'MESA';
      T     DBD [AR2, P#1.0];
      L     ']';
      T     DBB [AR2, P#5.0];
      +AR2  P#6.0;

      L     "DB812_UTs_Control".UT[#NumeroUT].MesaActual;
      T     #Valor;

// --- Convertir Valor a ASCII -  Mesa Actual
      TAR2;
      SRD   3;
      T     #NumBytes;  // Miro que offset tiene la String

      CALL  "FC893_Obtener_StringDelAtributo"
      ( DB_String := #NumDBEventos,
        OffsetIni := #NumBytes,
        Valor     := #Valor,
        OffsetFin := #Offset
      );  // Llamo a ObtenerStrinAtributo

      L     #Offset;
      SLD   3;
      LAR2;  // Recupero que offset tiene la String

// --- Ya esta convertido el Valor a ASCI - Fin Mesa Actual


////////////////////////////////////////////////////////////////////////////////
      OPN   DB [#DBEventos];
      L     '[';  // Evento - Atributo Motivo '[MOTI]'
      T     DBB [AR2, P#0.0];
      L     'MOTI';
      T     DBD [AR2, P#1.0];
      L     ']';
      T     DBB [AR2, P#5.0];
      +AR2  P#6.0;

      L     #EventoUT;  // Poner Motivo
      T     #Convertir;
      CALL  "FC895_Obtener_EtiquetaDeValor"
      ( ValorEvento    := #Convertir,
        EtiquetaEvento := #Conversion
      );

      OPN   DB [#DBEventos];
      L     #Conversion;
      T     DBD [AR2, P#0.0];
      +AR2  P#4.0;


////////////////////////////////////////////////////////////////////////////////
// --- Final del Formateo del Evento ---

      OPN   DB [#DBEventos];  // DB de Eventos Generados (A Emitir)
      L     '}';  // Fin de Evento '}'
      T     DBB [AR2, P#0.0];
      +AR2  P#1.0;


////////////////////////////////////////////////////////////////////////////////
////////////////////////////////////////////////////////////////////////////////
////////////////////////////////////////////////////////////////////////////////
// Dar por formateado el Evento

      L     0;  // 0 - Dar por Tratado
      T     "DB812_UTs_Control".UT[#NumeroUT].EstadoEventoAGenerar;

////////////////////////////////////////////////////////////////////////////////
/// Hay que Pedir Datos
      SET;
      AN    "DB812_UTs_Control".UT[#NumeroUT].AtributosDeLaUT.PeticionDeDatos;
      JC    NoPedirDatos_RUT_EventosUT;

      L     141;
      T     "DB812_UTs_Control".UT[#NumeroUT].EstadoEventoAGenerar;

NoPedirDatos_RUT_EventosUT:NOP   0;


////////////////////////////////////////////////////////////////////////////////
      JU    FinBucles_EventosUT;


// Fin del Evento RUT?
////////////////////////////////////////////////////////////////////////////////
////////////////////////////////////////////////////////////////////////////////
////////////////////////////////////////////////////////////////////////////////



NETWORK
TITLE = ---- Eventos de UT - Ausencia de la Mesa - RET!
GenerarEvento_RET_EventosUT:NOP   0;

////////////////////////////////////////////////////////////////////////////////
////////////////////////////////////////////////////////////////////////////////
////////////////////////////////////////////////////////////////////////////////
////////////////////////////////////////////////////////////////////////////////
// -- Formateo del Evento RET! - Ausencia de la Mesa

      L     #P_Eventos;
      LAR2;  // Puntero al DB de Eventos Generados

      TAR2;  // Mirar si es el primer evento de la lista
      L     0;
      ==I;
      JC    InicioBuffer_RET_EventosUT;  // Es el primero

      OPN   DB [#DBEventos];  // Hay que añadir si no es el primer evento
      L     ',';  // Separador entre eventos ','
      T     DBB [AR2, P#0.0];
      +AR2  P#1.0;

InicioBuffer_RET_EventosUT:NOP   0;
      OPN   DB [#DBEventos];  // DB de Eventos Generados (A Emitir)
      L     '{';  // Inicio de Evento '{'
      T     DBB [AR2, P#0.0];
      +AR2  P#1.0;

      L     'RET!';  // Evento 'RET!'
      T     DBD [AR2, P#0.0];
      +AR2  P#4.0;


////////////////////////////////////////////////////////////////////////////////
      L     '[';  // Evento - Atributo Mckey '[MCKY]'
      T     DBB [AR2, P#0.0];
      L     'MCKY';
      T     DBD [AR2, P#1.0];
      L     ']';
      T     DBB [AR2, P#5.0];
      +AR2  P#6.0;

      L     "DB812_UTs_Control".UT[#NumeroUT].Mckey;
      T     #Valor;

// --- Convertir Valor a ASCII - Mckey
      TAR2;
      SRD   3;
      T     #NumBytes;  // Miro que offset tiene la String

      CALL  "FC893_Obtener_StringDelAtributo"
      ( DB_String := #NumDBEventos,
        OffsetIni := #NumBytes,
        Valor     := #Valor,
        OffsetFin := #Offset
      );  // Llamo a ObtenerStrinAtributo

      L     #Offset;
      SLD   3;
      LAR2;  // Recupero que offset tiene la String

// --- Ya esta convertido el Valor a ASCI - Fin Mckey


////////////////////////////////////////////////////////////////////////////////
      OPN   DB [#DBEventos];
      L     '[';  // Evento - Atributo Mesa Actual '[MESA]'
      T     DBB [AR2, P#0.0];
      L     'MESA';
      T     DBD [AR2, P#1.0];
      L     ']';
      T     DBB [AR2, P#5.0];
      +AR2  P#6.0;

      L     "DB812_UTs_Control".UT[#NumeroUT].MesaActual;
      T     #Valor;

// --- Convertir Valor a ASCII -  Mesa Actual
      TAR2;
      SRD   3;
      T     #NumBytes;  // Miro que offset tiene la String

      CALL  "FC893_Obtener_StringDelAtributo"
      ( DB_String := #NumDBEventos,
        OffsetIni := #NumBytes,
        Valor     := #Valor,
        OffsetFin := #Offset
      );  // Llamo a ObtenerStrinAtributo

      L     #Offset;
      SLD   3;
      LAR2;  // Recupero que offset tiene la String

// --- Ya esta convertido el Valor a ASCI - Fin Mesa Actual


////////////////////////////////////////////////////////////////////////////////
// --- Final del Formato del Evento ---

      OPN   DB [#DBEventos];  // DB de Eventos Generados (A Emitir)
      L     '}';  // Fin de Evento '}'
      T     DBB [AR2, P#0.0];
      +AR2  P#1.0;


////////////////////////////////////////////////////////////////////////////////
////////////////////////////////////////////////////////////////////////////////
////////////////////////////////////////////////////////////////////////////////
////////////////////////////////////////////////////////////////////////////////
// Dar por formateado el Evento

      L     0;  // 0 - Dar por Tratado
      T     "DB812_UTs_Control".UT[#NumeroUT].EstadoEventoAGenerar;

      JU    FinBucles_EventosUT;

// Fin del formateo del Evento RET!
////////////////////////////////////////////////////////////////////////////////
////////////////////////////////////////////////////////////////////////////////
////////////////////////////////////////////////////////////////////////////////
////////////////////////////////////////////////////////////////////////////////



NETWORK
TITLE = ---- Evento de UT - Borrar la UT de la Mesa - BOR!
GenerarEvento_BOR_EventosUT:NOP   0;

////////////////////////////////////////////////////////////////////////////////
////////////////////////////////////////////////////////////////////////////////
////////////////////////////////////////////////////////////////////////////////
////////////////////////////////////////////////////////////////////////////////
// -- Formateo del Evento BOR! - Borrada UT del Sistema


      L     #P_Eventos;
      LAR2;  // Puntero al DB de Eventos Generados

      TAR2;  // Mirar si es el primer evento de la lista
      L     0;
      ==I;
      JC    InicioBuffer_BOR_EventosUT;  // Es el primero

      OPN   DB [#DBEventos];  // Hay que añadir si no es el primer evento
      L     ',';  // Separador entre eventos ','
      T     DBB [AR2, P#0.0];
      +AR2  P#1.0;

InicioBuffer_BOR_EventosUT:NOP   0;
      OPN   DB [#DBEventos];  // DB de Eventos Generados (A Emitir)
      L     '{';  // Inicio de Evento '{'
      T     DBB [AR2, P#0.0];
      +AR2  P#1.0;

      L     'BOR!';  // Evento 'BOR!'
      T     DBD [AR2, P#0.0];
      +AR2  P#4.0;


////////////////////////////////////////////////////////////////////////////////
      L     '[';  // Evento - Atributo Mckey '[MCKY]'
      T     DBB [AR2, P#0.0];
      L     'MCKY';
      T     DBD [AR2, P#1.0];
      L     ']';
      T     DBB [AR2, P#5.0];
      +AR2  P#6.0;

      L     "DB812_UTs_Control".UT[#NumeroUT].Mckey;
      T     #Valor;

// --- Convertir Valor a ASCII - Mckey
      TAR2;
      SRD   3;
      T     #NumBytes;  // Miro que offset tiene la String

      CALL  "FC893_Obtener_StringDelAtributo"
      ( DB_String := #NumDBEventos,
        OffsetIni := #NumBytes,
        Valor     := #Valor,
        OffsetFin := #Offset
      );  // Llamo a ObtenerStrinAtributo

      L     #Offset;
      SLD   3;
      LAR2;  // Recupero que offset tiene la String

// --- Ya esta convertido el Valor a ASCI - Fin Mckey


////////////////////////////////////////////////////////////////////////////////
      OPN   DB [#DBEventos];
      L     '[';  // Evento - Atributo Mesa Actual 'MESA'
      T     DBB [AR2, P#0.0];
      L     'MESA';
      T     DBD [AR2, P#1.0];
      L     ']';
      T     DBB [AR2, P#5.0];
      +AR2  P#6.0;

      L     "DB812_UTs_Control".UT[#NumeroUT].MesaActual;
      T     #Valor;

// --- Convertir Valor a ASCII -  Mesa Actual
      TAR2;
      SRD   3;
      T     #NumBytes;  // Miro que offset tiene la String

      CALL  "FC893_Obtener_StringDelAtributo"
      ( DB_String := #NumDBEventos,
        OffsetIni := #NumBytes,
        Valor     := #Valor,
        OffsetFin := #Offset
      );  // Llamo a ObtenerStrinAtributo

      L     #Offset;
      SLD   3;
      LAR2;  // Recupero que offset tiene la String

// --- Ya esta convertido el Valor a ASCI - Fin Mesa Actual


////////////////////////////////////////////////////////////////////////////////
// --- Final del Formato del Evento ---

      OPN   DB [#DBEventos];  // DB de Eventos Generados (A Emitir)
      L     '}';  // Fin de Evento '}'
      T     DBB [AR2, P#0.0];
      +AR2  P#1.0;


////////////////////////////////////////////////////////////////////////////////
////////////////////////////////////////////////////////////////////////////////
////////////////////////////////////////////////////////////////////////////////
////////////////////////////////////////////////////////////////////////////////
// Borrar la UT de la Base de datos

      CALL  "FC722_EliminarUT_DeMesa"
      ( NumeroUT := #NumeroUT
      );

      JU    FinBucles_EventosUT;

// Fin del formateo del Evento BOR!
////////////////////////////////////////////////////////////////////////////////
////////////////////////////////////////////////////////////////////////////////
////////////////////////////////////////////////////////////////////////////////
////////////////////////////////////////////////////////////////////////////////



NETWORK
TITLE = ---- Evento de UT - Nueva UT en la Mesa - NUUT
GenerarEvento_NUUT_EventosUT:NOP   0;

////////////////////////////////////////////////////////////////////////////////
////////////////////////////////////////////////////////////////////////////////
////////////////////////////////////////////////////////////////////////////////
////////////////////////////////////////////////////////////////////////////////
// -- Formateo del Evento NUUT - Nueva UT en la Mesa

      L     #P_Eventos;
      LAR2;  // Puntero al DB de Eventos Generados

      TAR2;  // Mirar si es el primer evento de la lista
      L     0;
      ==I;
      JC    InicioBuffer_NUUT_EventosUT;  // Es el primero

      OPN   DB [#DBEventos];  // Hay que añadir si no es el primer evento
      L     ',';  // Separador entre eventos ','
      T     DBB [AR2, P#0.0];
      +AR2  P#1.0;

InicioBuffer_NUUT_EventosUT:NOP   0;
      OPN   DB [#DBEventos];  // DB de Eventos Generados (A Emitir)
      L     '{';  // Inicio de Evento '{'
      T     DBB [AR2, P#0.0];
      +AR2  P#1.0;

      L     'NUUT';  // Evento  'NUUT'
      T     DBD [AR2, P#0.0];
      +AR2  P#4.0;


////////////////////////////////////////////////////////////////////////////////
      OPN   DB [#DBEventos];
      L     '[';  // Evento - Atributo Mesa Actual '[MESA]'
      T     DBB [AR2, P#0.0];
      L     'MESA';
      T     DBD [AR2, P#1.0];
      L     ']';
      T     DBB [AR2, P#5.0];
      +AR2  P#6.0;

      L     "DB812_UTs_Control".UT[#NumeroUT].MesaActual;
      T     #Valor;

// --- Convertir Valor a ASCII -  Mesa Actual
      TAR2;
      SRD   3;
      T     #NumBytes;  // Miro que offset tiene la String

      CALL  "FC893_Obtener_StringDelAtributo"
      ( DB_String := #NumDBEventos,
        OffsetIni := #NumBytes,
        Valor     := #Valor,
        OffsetFin := #Offset
      );  // Llamo a ObtenerStrinAtributo

      L     #Offset;
      SLD   3;
      LAR2;  // Recupero que offset tiene la String

// --- Ya esta convertido el Valor a ASCI - Fin Mesa Actual


////////////////////////////////////////////////////////////////////////////////
////////////////////////////////////////////////////////////////////////////////
////////////////////////////////////////////////////////////////////////////////
////////////////////////////////////////////////////////////////////////////////
// --- Caracteristicas de la UT a Emitir


////////////////////////////////////////////////////////////////////////////////
// --- Atributo de ALTURA COTA (Si es necesario) ---
      SET;
      AN    "DB850_DefinicionMesas".Mesa[#NumMesa].AtributosGalibo_DeEvento.Cota_Altura;  // Tiene Cota Altura ?
      JC    CotaAltura_NUNUT_EventosUT;

      L     "DB815_UTs_Datos".UT[#NumeroUT].CotaAltura;
      T     #Valor;

      OPN   DB [#DBEventos];
      L     '[';  // Evento - Atributo Altura Cota '[ALTO]'
      T     DBB [AR2, P#0.0];
      L     'COTA';
      T     DBD [AR2, P#1.0];
      L     ']';
      T     DBB [AR2, P#5.0];
      +AR2  P#6.0;

// --- Convertir Valor a ASCII -  Altura Cota
      TAR2;
      SRD   3;
      T     #NumBytes;  // Miro que offset tiene la String

      CALL  "FC893_Obtener_StringDelAtributo"
      ( DB_String := #NumDBEventos,
        OffsetIni := #NumBytes,
        Valor     := #Valor,
        OffsetFin := #Offset
      );  // Llamo a ObtenerStrinAtributo

      L     #Offset;
      SLD   3;
      LAR2;  // Recupero que offset tiene la String

// --- Ya esta convertido el Valor a ASCI - Fin Altura Cota
CotaAltura_NUNUT_EventosUT:NOP   0;


////////////////////////////////////////////////////////////////////////////////
////////////////////////////////////////////////////////////////////////////////
////////////////////////////////////////////////////////////////////////////////
////////////////////////////////////////////////////////////////////////////////
// --- Atributo de GALIBO (ALTO, ANCH, LARG, REMO) (Si es necesario) ---
      SET;
      AN    "DB850_DefinicionMesas".Mesa[#NumMesa].AtributosGalibo_DeEvento.Altura;  // Tiene Altura ?
      JC    CodigoAltura_NUUT_EventosUT;

      OPN   DB [#DBEventos];
      L     '[';  // Evento - Atributo Galibo Altura '[ALTO]'
      T     DBB [AR2, P#0.0];
      L     'ALTO';
      T     DBD [AR2, P#1.0];
      L     ']';
      T     DBB [AR2, P#5.0];
      +AR2  P#6.0;

      L     "DB815_UTs_Datos".UT[#NumeroUT].GaliboAltura;
      T     #Valor;

// --- Convertir Valor a ASCII -  Alto
      TAR2;
      SRD   3;
      T     #NumBytes;  // Miro que offset tiene la String

      CALL  "FC893_Obtener_StringDelAtributo"
      ( DB_String := #NumDBEventos,
        OffsetIni := #NumBytes,
        Valor     := #Valor,
        OffsetFin := #Offset
      );  // Llamo a ObtenerStrinAtributo

      L     #Offset;
      SLD   3;
      LAR2;  // Recupero que offset tiene la String

// nieves inicio modificación emisión atributo VACI

//Comprobar si tenemos que emitir el evento

      SET;
      L     "DB815_UTs_Datos".UT[#NumeroUT].GaliboVacia;
      L     0;
      ==I;
      JC    CodigoAltura_NUUT_EventosUT;

      OPN   DB [#DBEventos];
      L     '[';  // Evento - Atributo Galibo Altura '[ALTO]'
      T     DBB [AR2, P#0.0];
      L     'VACI';
      T     DBD [AR2, P#1.0];
      L     ']';
      T     DBB [AR2, P#5.0];
      +AR2  P#6.0;

      L     "DB815_UTs_Datos".UT[#NumeroUT].GaliboVacia;
      L     1;
      -I;
      T     #Valor;

// --- Convertir Valor a ASCII -  VACIO
      TAR2;
      SRD   3;
      T     #NumBytes;  // Miro que offset tiene la String

      CALL  "FC893_Obtener_StringDelAtributo"
      ( DB_String := #NumDBEventos,
        OffsetIni := #NumBytes,
        Valor     := #Valor,
        OffsetFin := #Offset
      );  // Llamo a ObtenerStrinAtributo


      L     #Offset;
      SLD   3;
      LAR2;  // Recupero que offset tiene la String


// fin modificación atributo VACI

// --- Ya esta convertido el Valor a ASCI - Fin Alto
CodigoAltura_NUUT_EventosUT:NOP   0;


////////////////////////////////////////////////////////////////////////////////
      SET;
      AN    "DB850_DefinicionMesas".Mesa[#NumMesa].AtributosGalibo_DeEvento.Anchura;  // Tiene Anchura ?
      JC    CodigoAnchura_NUUT_EventosUT;

      OPN   DB [#DBEventos];
      L     '[';  // Evento - Atributo Galibo Anchura '[ANCH]'
      T     DBB [AR2, P#0.0];
      L     'ANCH';
      T     DBD [AR2, P#1.0];
      L     ']';
      T     DBB [AR2, P#5.0];
      +AR2  P#6.0;

      L     "DB815_UTs_Datos".UT[#NumeroUT].GaliboAnchura;
      T     #Valor;

// --- Convertir Valor a ASCII -  Anchura
      TAR2;
      SRD   3;
      T     #NumBytes;  // Miro que offset tiene la String

      CALL  "FC893_Obtener_StringDelAtributo"
      ( DB_String := #NumDBEventos,
        OffsetIni := #NumBytes,
        Valor     := #Valor,
        OffsetFin := #Offset
      );  // Llamo a ObtenerStrinAtributo

      L     #Offset;
      SLD   3;
      LAR2;  // Recupero que offset tiene la String

// --- Ya esta convertido el Valor a ASCI - Fin Anchura
CodigoAnchura_NUUT_EventosUT:NOP   0;


////////////////////////////////////////////////////////////////////////////////
      SET;
      AN    "DB850_DefinicionMesas".Mesa[#NumMesa].AtributosGalibo_DeEvento.Profundidad;  // Tiene Profundidad ?
      JC    CodigoLargura_NUUT_EventosUT;

      OPN   DB [#DBEventos];
      L     '[';  // Evento - Atributo Galibo Profuncidad '[PROF]'
      T     DBB [AR2, P#0.0];
      L     'PROF';
      T     DBD [AR2, P#1.0];
      L     ']';
      T     DBB [AR2, P#5.0];
      +AR2  P#6.0;

      L     "DB815_UTs_Datos".UT[#NumeroUT].GaliboProfundidad;
      T     #Valor;

// --- Convertir Valor a ASCII -  Profundidad
      TAR2;
      SRD   3;
      T     #NumBytes;  // Miro que offset tiene la String

      CALL  "FC893_Obtener_StringDelAtributo"
      ( DB_String := #NumDBEventos,
        OffsetIni := #NumBytes,
        Valor     := #Valor,
        OffsetFin := #Offset
      );  // Llamo a ObtenerStrinAtributo

      L     #Offset;
      SLD   3;
      LAR2;  // Recupero que offset tiene la String

// --- Ya esta convertido el Valor a ASCI - Fin Profundidad
CodigoLargura_NUUT_EventosUT:NOP   0;


////////////////////////////////////////////////////////////////////////////////
      SET;
      AN    "DB850_DefinicionMesas".Mesa[#NumMesa].AtributosGalibo_DeEvento.Remontado;  // Tiene Remontado ?
      JC    CodigoRemontado_NUUT_EventosUT;

      OPN   DB [#DBEventos];
      L     '[';  // Evento - Atributo Galibo Remontada '[REMO]'
      T     DBB [AR2, P#0.0];
      L     'REMO';
      T     DBD [AR2, P#1.0];
      L     ']';
      T     DBB [AR2, P#5.0];
      +AR2  P#6.0;

      L     "DB815_UTs_Datos".UT[#NumeroUT].GaliboRemontada;
      L     1;
      -I;
      L     W#16#30;
      +I;
      OPN   DB [#DBEventos];
      T     DBB [AR2, P#0.0];
      +AR2  P#1.0;

CodigoRemontado_NUUT_EventosUT:NOP   0;

////////////////////////////////////////////////////////////////////////////////
////////////////////////////////////////////////////////////////////////////////
////////////////////////////////////////////////////////////////////////////////
////////////////////////////////////////////////////////////////////////////////


////////////////////////////////////////////////////////////////////////////////
// --- Atributo de PESO (Si es necesario) ---
      SET;
      AN    "DB850_DefinicionMesas".Mesa[#NumMesa].AtributosGalibo_DeEvento.Peso;  // Tiene Peso ?
      JC    Peso_NUUT_EventoUT;

      L     "DB815_UTs_Datos".UT[#NumeroUT].Peso;
      T     #Valor;

      OPN   DB [#DBEventos];
      L     '[';  // Evento - Atributo Peso '[PESO]'
      T     DBB [AR2, P#0.0];
      L     'PESO';
      T     DBD [AR2, P#1.0];
      L     ']';
      T     DBB [AR2, P#5.0];
      +AR2  P#6.0;

// --- Convertir Valor a ASCII -  Peso
      TAR2;
      SRD   3;
      T     #NumBytes;  // Miro que offset tiene la String

      CALL  "FC893_Obtener_StringDelAtributo"
      ( DB_String := #NumDBEventos,
        OffsetIni := #NumBytes,
        Valor     := #Valor,
        OffsetFin := #Offset
      );  // Llamo a ObtenerStrinAtributo

      L     #Offset;
      SLD   3;
      LAR2;  // Recupero que offset tiene la String

// --- Ya esta convertido el Valor a ASCI - Fin Peso
Peso_NUUT_EventoUT:NOP   0;


////////////////////////////////////////////////////////////////////////////////
// --- Atributo de ANCHURA COTA (Si es necesario) ---
      SET;
      AN    "DB850_DefinicionMesas".Mesa[#NumMesa].AtributosGalibo_DeEvento.Cota_Anchura;  // Tiene Cota de Anchura ?
      JC    CotaAnchura_NUUT_EventoUT;

      L     "DB815_UTs_Datos".UT[#NumeroUT].CotaAnchura;
      T     #Valor;

      OPN   DB [#DBEventos];
      L     '[';  // Evento - Atributo Anchura Cota '[COTW]'
      T     DBB [AR2, P#0.0];
      L     'COTW';
      T     DBD [AR2, P#1.0];
      L     ']';
      T     DBB [AR2, P#5.0];
      +AR2  P#6.0;

// --- Convertir Valor a ASCII -  Anchura Cota
      TAR2;
      SRD   3;
      T     #NumBytes;  // Miro que offset tiene la String

      CALL  "FC893_Obtener_StringDelAtributo"
      ( DB_String := #NumDBEventos,
        OffsetIni := #NumBytes,
        Valor     := #Valor,
        OffsetFin := #Offset
      );  // Llamo a ObtenerStrinAtributo

      L     #Offset;
      SLD   3;
      LAR2;  // Recupero que offset tiene la String

// --- Ya esta convertido el Valor a ASCI - Fin Anchura Cota
CotaAnchura_NUUT_EventoUT:NOP   0;


////////////////////////////////////////////////////////////////////////////////
// --- Atributo de LARGURA COTA (Si es necesario) ---
      SET;
      AN    "DB850_DefinicionMesas".Mesa[#NumMesa].AtributosGalibo_DeEvento.Cota_Profundidad;  // Tiene Cota de Profundidad ?
      JC    CotaLargura_NUUT_EventoUT;

      L     "DB815_UTs_Datos".UT[#NumeroUT].CotaProfundidad;
      T     #Valor;

      OPN   DB [#DBEventos];
      L     '[';  // Evento - Atributo Largura Cota '[COTL]'
      T     DBB [AR2, P#0.0];
      L     'COTL';
      T     DBD [AR2, P#1.0];
      L     ']';
      T     DBB [AR2, P#5.0];
      +AR2  P#6.0;

// --- Convertir Valor a ASCII -  Largura Cota
      TAR2;
      SRD   3;
      T     #NumBytes;  // Miro que offset tiene la String

      CALL  "FC893_Obtener_StringDelAtributo"
      ( DB_String := #NumDBEventos,
        OffsetIni := #NumBytes,
        Valor     := #Valor,
        OffsetFin := #Offset
      );  // Llamo a ObtenerStrinAtributo

      L     #Offset;
      SLD   3;
      LAR2;  // Recupero que offset tiene la String

// --- Ya esta convertido el Valor a ASCI - Fin Largura Cota
CotaLargura_NUUT_EventoUT:NOP   0;


////////////////////////////////////////////////////////////////////////////////
////////////////////////////////////////////////////////////////////////////////
////////////////////////////////////////////////////////////////////////////////
////////////////////////////////////////////////////////////////////////////////
// --- Atributo de TIPO, HUECO y TACO (Si es necesario) ---
      SET;  // Tiene Taco ?
      AN    "DB850_DefinicionMesas".Mesa[#NumMesa].AtributosGalibo_DeEvento.Taco;
      JC    CodigoTaco_NUUT_EventosUT;

      OPN   DB [#DBEventos];
      L     '[';  // Evento - Atributo Galibo Taco '[TACO]'
      T     DBB [AR2, P#0.0];
      L     'TACO';
      T     DBD [AR2, P#1.0];
      L     ']';
      T     DBB [AR2, P#5.0];
      +AR2  P#6.0;

      L     "DB815_UTs_Datos".UT[#NumeroUT].GaliboTaco;
      T     #Valor;

// --- Convertir Valor a ASCII -  Taco
      TAR2;
      SRD   3;
      T     #NumBytes;  // Miro que offset tiene la String

      CALL  "FC893_Obtener_StringDelAtributo"
      ( DB_String := #NumDBEventos,
        OffsetIni := #NumBytes,
        Valor     := #Valor,
        OffsetFin := #Offset
      );  // Llamo a ObtenerStrinAtributo

      L     #Offset;
      SLD   3;
      LAR2;  // Recupero que offset tiene la String

// --- Ya esta convertido el Valor a ASCI - Fin Taco
CodigoTaco_NUUT_EventosUT:NOP   0;


////////////////////////////////////////////////////////////////////////////////
      SET;  // Tiene Hueco ?
      AN    "DB850_DefinicionMesas".Mesa[#NumMesa].AtributosGalibo_DeEvento.Hueco;
      JC    CodigoHueco_NUUT_EventosUT;

      OPN   DB [#DBEventos];
      L     '[';  // Evento - Atributo Galibo Hueco '[HUEC]'
      T     DBB [AR2, P#0.0];
      L     'HUEC';
      T     DBD [AR2, P#1.0];
      L     ']';
      T     DBB [AR2, P#5.0];
      +AR2  P#6.0;

      L     "DB815_UTs_Datos".UT[#NumeroUT].GaliboHueco;
      T     #Valor;

// --- Convertir Valor a ASCII -  Hueco
      TAR2;
      SRD   3;
      T     #NumBytes;  // Miro que offset tiene la String

      CALL  "FC893_Obtener_StringDelAtributo"
      ( DB_String := #NumDBEventos,
        OffsetIni := #NumBytes,
        Valor     := #Valor,
        OffsetFin := #Offset
      );  // Llamo a ObtenerStrinAtributo

      L     #Offset;
      SLD   3;
      LAR2;  // Recupero que offset tiene la String

// --- Ya esta convertido el Valor a ASCI - Fin Hueco
CodigoHueco_NUUT_EventosUT:NOP   0;


////////////////////////////////////////////////////////////////////////////////
      SET;  // Tiene Hueco R ?
      AN    "DB850_DefinicionMesas".Mesa[#NumMesa].AtributosGalibo_DeEvento.HuecoRemontado;
      JC    CodigoHuecoR_NUUT_EventosUT;

      OPN   DB [#DBEventos];
      L     '[';  // Evento - Atributo Galibo Hueco '[HUEC]'
      T     DBB [AR2, P#0.0];
      L     'HUER';
      T     DBD [AR2, P#1.0];
      L     ']';
      T     DBB [AR2, P#5.0];
      +AR2  P#6.0;

      L     "DB815_UTs_Datos".UT[#NumeroUT].GaliboHuecoRemontado;
      T     #Valor;

// --- Convertir Valor a ASCII -  Huer
      TAR2;
      SRD   3;
      T     #NumBytes;  // Miro que offset tiene la String

      CALL  "FC893_Obtener_StringDelAtributo"
      ( DB_String := #NumDBEventos,
        OffsetIni := #NumBytes,
        Valor     := #Valor,
        OffsetFin := #Offset
      );  // Llamo a ObtenerStrinAtributo

      L     #Offset;
      SLD   3;
      LAR2;  // Recupero que offset tiene la String

// --- Ya esta convertido el Valor a ASCI - Fin Huer
CodigoHuecoR_NUUT_EventosUT:NOP   0;


////////////////////////////////////////////////////////////////////////////////
      SET;  // Tiene Tipo ?
      AN    "DB850_DefinicionMesas".Mesa[#NumMesa].AtributosGalibo_DeEvento.Tipo;
      JC    CodigoTipo_NUUT_EventosUT;

      OPN   DB [#DBEventos];
      L     '[';  // Evento - Atributo Galibo Hueco '[HUEC]'
      T     DBB [AR2, P#0.0];
      L     'TIPO';
      T     DBD [AR2, P#1.0];
      L     ']';
      T     DBB [AR2, P#5.0];
      +AR2  P#6.0;

      L     "DB815_UTs_Datos".UT[#NumeroUT].GaliboTipoCarga;
      L     W#16#F;
      <>I;
      JC    CodigoTipoExiste_NUUT_EventosUT;

      OPN   DB [#DBEventos];
      L     'ERRO';
      T     DBD [AR2, P#0.0];
      +AR2  P#4.0;

      JU    CodigoTipo_NUUT_EventosUT;

CodigoTipoExiste_NUUT_EventosUT:NOP   0;
      L     "DB815_UTs_Datos".UT[#NumeroUT].GaliboTipoCarga;
      L     3000;
      +I;
      T     #Convertir;
      CALL  "FC895_Obtener_EtiquetaDeValor"
      ( ValorEvento    := #Convertir,
        EtiquetaEvento := #Conversion
      );

      OPN   DB [#DBEventos];
      L     #Conversion;
      T     DBD [AR2, P#0.0];
      +AR2  P#4.0;

CodigoTipo_NUUT_EventosUT:NOP   0;

////////////////////////////////////////////////////////////////////////////////
////////////////////////////////////////////////////////////////////////////////
////////////////////////////////////////////////////////////////////////////////
////////////////////////////////////////////////////////////////////////////////


////////////////////////////////////////////////////////////////////////////////
////////////////////////////////////////////////////////////////////////////////
////////////////////////////////////////////////////////////////////////////////
////////////////////////////////////////////////////////////////////////////////
// --- Atributo de COLOR (Si es necesario) ---
      SET;  // Tiene Color ?
      AN    "DB850_DefinicionMesas".Mesa[#NumMesa].AtributosGalibo_DeEvento.Color;
      JC    CodigoColor_NUUT_EventosUT;

      OPN   DB [#DBEventos];
      L     '[';  // Evento - Atributo Galibo Hueco '[HUEC]'
      T     DBB [AR2, P#0.0];
      L     'COLO';
      T     DBD [AR2, P#1.0];
      L     ']';
      T     DBB [AR2, P#5.0];
      +AR2  P#6.0;

      L     "DB815_UTs_Datos".UT[#NumeroUT].GaliboColor;
      L     W#16#F;
      <>I;
      JC    CodigoColorExiste_NUUT_EventosUT;

      OPN   DB [#DBEventos];
      L     'ERRO';  // ERROR De COLOR
      T     DBD [AR2, P#0.0];
      +AR2  P#4.0;

      JU    CodigoColor_NUUT_EventosUT;

CodigoColorExiste_NUUT_EventosUT:NOP   0;
      L     "DB815_UTs_Datos".UT[#NumeroUT].GaliboColor;
      L     3100;
      +I;
      T     #Convertir;
      CALL  "FC895_Obtener_EtiquetaDeValor"
      ( ValorEvento    := #Convertir,
        EtiquetaEvento := #Conversion
      );

      OPN   DB [#DBEventos];
      L     #Conversion;
      T     DBD [AR2, P#0.0];
      +AR2  P#4.0;

CodigoColor_NUUT_EventosUT:NOP   0;


////////////////////////////////////////////////////////////////////////////////
      SET;
      AN    "DB850_DefinicionMesas".Mesa[#NumMesa].AtributosGalibo_DeEvento.Patin;
      JC    CodigoPatin_NUUT_EventosUT;  // Tiene Patin ?

      OPN   DB [#DBEventos];
      L     '[';  // Evento - Atributo Galibo Patin '[PATI]'
      T     DBB [AR2, P#0.0];
      L     'PATI';
      T     DBD [AR2, P#1.0];
      L     ']';
      T     DBB [AR2, P#5.0];
      +AR2  P#6.0;

      L     "DB815_UTs_Datos".UT[#NumeroUT].GaliboPatin;
      T     #Valor;

// --- Convertir Valor a ASCII -  Patin
      TAR2;
      SRD   3;
      T     #NumBytes;  // Miro que offset tiene la String

      CALL  "FC893_Obtener_StringDelAtributo"
      ( DB_String := #NumDBEventos,
        OffsetIni := #NumBytes,
        Valor     := #Valor,
        OffsetFin := #Offset
      );  // Llamo a ObtenerStrinAtributo

